C09151=1184.865,-10.764,-44.192,179.961,5.758,149.033
C09152=1184.870,-11.013,-44.179,179.959,5.759,149.034
C09153=1184.875,-11.263,-44.165,179.956,5.758,149.035
C09154=1184.880,-11.512,-44.153,179.953,5.758,149.035
C09155=1184.886,-11.762,-44.139,179.951,5.757,149.036
C09156=1184.891,-12.012,-44.126,179.949,5.756,149.036
C09157=1184.896,-12.261,-44.112,179.946,5.756,149.037
C09158=1184.901,-12.511,-44.099,179.944,5.755,149.038
C09159=1184.907,-12.760,-44.086,179.941,5.755,149.038
C09160=1184.911,-13.010,-44.073,179.938,5.754,149.039
C09161=1184.916,-13.260,-44.061,179.936,5.754,149.040
C09162=1184.922,-13.509,-44.047,179.934,5.754,149.040
C09163=1184.926,-13.759,-44.034,179.932,5.753,149.041
C09164=1184.932,-14.008,-44.021,179.929,5.753,149.041
C09165=1184.937,-14.258,-44.008,179.926,5.752,149.042
C09166=1184.942,-14.508,-43.995,179.924,5.751,149.043
C09167=1184.947,-14.757,-43.981,179.921,5.751,149.043
C09168=1184.952,-15.007,-43.968,179.919,5.751,149.044
C09169=1184.957,-15.256,-43.956,179.916,5.750,149.045
C09170=1184.963,-15.506,-43.942,179.914,5.749,149.045
C09171=1184.967,-15.756,-43.929,179.912,5.750,149.046
C09172=1184.973,-16.005,-43.916,179.909,5.749,149.047
C09173=1184.978,-16.255,-43.903,179.907,5.748,149.047
C09174=1184.983,-16.504,-43.890,179.904,5.748,149.048
C09175=1184.988,-16.754,-43.877,179.902,5.747,149.048
C09176=1184.993,-17.004,-43.864,179.899,5.747,149.049
C09177=1184.998,-17.253,-43.851,179.897,5.746,149.050
C09178=1185.004,-17.503,-43.838,179.894,5.746,149.050
C09179=1185.008,-17.753,-43.825,179.892,5.746,149.051
C09180=1185.014,-18.002,-43.812,179.890,5.745,149.052
C09181=1185.019,-18.251,-43.800,179.887,5.745,149.052
C09182=1185.024,-18.502,-43.786,179.885,5.744,149.053
C09183=1185.029,-18.751,-43.774,179.882,5.744,149.054
C09184=1185.034,-19.000,-43.761,179.880,5.743,149.054
C09185=1185.039,-19.251,-43.747,179.877,5.742,149.055
C09186=1185.045,-19.500,-43.735,179.875,5.742,149.055
C09187=1185.050,-19.749,-43.722,179.872,5.742,149.056
C09188=1185.054,-19.999,-43.709,179.870,5.741,149.057
C09189=1185.060,-20.249,-43.696,179.868,5.741,149.057
C09190=1185.065,-20.498,-43.684,179.865,5.741,149.058
C09191=1185.070,-20.748,-43.671,179.862,5.740,149.059
C09192=1185.075,-20.998,-43.658,179.860,5.739,149.059
C09193=1185.081,-21.247,-43.645,179.857,5.739,149.060
C09194=1185.086,-21.497,-43.632,179.855,5.739,149.060
C09195=1185.090,-21.747,-43.619,179.853,5.739,149.061
C09196=1185.096,-21.996,-43.607,179.851,5.738,149.062
C09197=1185.101,-22.246,-43.593,179.848,5.737,149.062
C09198=1185.106,-22.495,-43.581,179.845,5.737,149.063
C09199=1185.111,-22.745,-43.568,179.843,5.736,149.063
C09200=1185.116,-22.994,-43.555,179.840,5.736,149.064
C09201=1185.122,-23.264,-43.541,179.838,5.735,149.065
C09202=1185.128,-23.534,-43.528,179.835,5.735,149.066
C09203=1185.134,-23.804,-43.514,179.832,5.734,149.066
C09204=1185.139,-24.074,-43.500,179.830,5.734,149.067
C09205=1185.144,-24.323,-43.488,179.828,5.734,149.068
C09206=1185.149,-24.572,-43.475,179.826,5.733,149.068
C09207=1185.154,-24.822,-43.463,179.823,5.733,149.069
C09208=1185.159,-25.072,-43.449,179.820,5.732,149.070
C09209=1185.165,-25.322,-43.437,179.818,5.732,149.070
C09210=1185.170,-25.571,-43.425,179.815,5.731,149.071
C09211=1185.175,-25.820,-43.412,179.813,5.732,149.071
C09212=1185.180,-26.070,-43.399,179.811,5.731,149.072
C09213=1185.184,-26.320,-43.386,179.808,5.731,149.073
C09214=1185.190,-26.569,-43.374,179.806,5.730,149.073
C09215=1185.195,-26.819,-43.362,179.803,5.729,149.074
C09216=1185.201,-27.069,-43.349,179.800,5.729,149.075
C09217=1185.206,-27.318,-43.336,179.799,5.729,149.075
C09218=1185.211,-27.568,-43.323,179.796,5.728,149.076
C09219=1185.216,-27.818,-43.311,179.794,5.728,149.077
C09220=1185.221,-28.067,-43.299,179.791,5.727,149.077
C09221=1185.226,-28.317,-43.286,179.789,5.727,149.078
C09222=1185.231,-28.566,-43.273,179.786,5.726,149.078
C09223=1185.236,-28.817,-43.261,179.784,5.727,149.079
C09224=1185.241,-29.066,-43.249,179.781,5.726,149.080
C09225=1185.246,-29.315,-43.236,179.779,5.725,149.080
C09226=1185.252,-29.565,-43.224,179.776,5.725,149.081
C09227=1185.257,-29.814,-43.212,179.774,5.724,149.082
C09228=1185.262,-30.064,-43.199,179.772,5.725,149.082
C09229=1185.267,-30.314,-43.186,179.770,5.724,149.083
C09230=1185.272,-30.564,-43.174,179.767,5.723,149.084
C09231=1185.277,-30.813,-43.161,179.764,5.723,149.084
C09232=1185.282,-31.062,-43.149,179.762,5.722,149.085
C09233=1185.288,-31.312,-43.137,179.759,5.722,149.085
C09234=1185.293,-31.562,-43.124,179.757,5.722,149.086
C09235=1185.298,-31.812,-43.112,179.755,5.722,149.087
C09236=1185.303,-32.062,-43.100,179.752,5.721,149.087
C09237=1185.308,-32.311,-43.087,179.750,5.720,149.088
C09238=1185.313,-32.561,-43.075,179.747,5.720,149.089
C09239=1185.318,-32.810,-43.062,179.745,5.720,149.089
C09240=1185.324,-33.060,-43.051,179.743,5.719,149.090
C09241=1185.329,-33.309,-43.038,179.740,5.719,149.091
C09242=1185.334,-33.559,-43.025,179.738,5.719,149.091
C09243=1185.340,-33.809,-43.013,179.735,5.718,149.092
C09244=1185.344,-34.059,-43.000,179.733,5.718,149.092
C09245=1185.350,-34.309,-42.989,179.731,5.718,149.093
C09246=1185.355,-34.558,-42.976,179.728,5.717,149.094
C09247=1185.360,-34.808,-42.964,179.726,5.716,149.094
C09248=1185.365,-35.057,-42.952,179.723,5.716,149.095
C09249=1185.371,-35.307,-42.940,179.721,5.716,149.096
C09250=1185.376,-35.556,-42.927,179.718,5.716,149.096
C09251=1185.381,-35.806,-42.915,179.716,5.715,149.097
C09252=1185.386,-36.056,-42.903,179.714,5.715,149.098
C09253=1185.392,-36.306,-42.891,179.712,5.715,149.098
C09254=1185.397,-36.555,-42.878,179.709,5.714,149.099
C09255=1185.402,-36.805,-42.867,179.707,5.714,149.099
C09256=1185.407,-37.054,-42.854,179.704,5.713,149.100
C09257=1185.412,-37.304,-42.842,179.701,5.713,149.101
C09258=1185.417,-37.553,-42.830,179.700,5.713,149.101
C09259=1185.422,-37.804,-42.817,179.697,5.712,149.102
C09260=1185.427,-38.053,-42.805,179.694,5.712,149.103
C09261=1185.433,-38.303,-42.793,179.692,5.711,149.103
C09262=1185.438,-38.552,-42.780,179.690,5.711,149.104
C09263=1185.442,-38.802,-42.769,179.688,5.711,149.105
C09264=1185.448,-39.052,-42.757,179.685,5.710,149.105
C09265=1185.453,-39.301,-42.745,179.683,5.710,149.106
C09266=1185.458,-39.551,-42.733,179.680,5.709,149.106
C09267=1185.464,-39.800,-42.720,179.678,5.710,149.107
C09268=1185.469,-40.050,-42.708,179.675,5.709,149.108
C09269=1185.474,-40.300,-42.697,179.673,5.708,149.108
C09270=1185.479,-40.549,-42.684,179.670,5.708,149.109
C09271=1185.484,-40.799,-42.672,179.668,5.707,149.110
C09272=1185.490,-41.049,-42.661,179.666,5.708,149.110
C09273=1185.495,-41.299,-42.648,179.663,5.707,149.111
C09274=1185.499,-41.548,-42.637,179.661,5.706,149.112
C09275=1185.505,-41.798,-42.625,179.658,5.706,149.112
C09276=1185.510,-42.047,-42.612,179.657,5.706,149.113
C09277=1185.515,-42.297,-42.600,179.654,5.706,149.113
C09278=1185.521,-42.547,-42.588,179.651,5.705,149.114
C09279=1185.525,-42.796,-42.576,179.649,5.705,149.115
C09280=1185.531,-43.046,-42.565,179.647,5.705,149.115
C09281=1185.536,-43.296,-42.553,179.644,5.704,149.116
C09282=1185.541,-43.545,-42.540,179.642,5.704,149.117
C09283=1185.546,-43.795,-42.529,179.639,5.703,149.117
C09284=1185.551,-44.045,-42.517,179.637,5.703,149.118
C09285=1185.557,-44.294,-42.505,179.635,5.703,149.119
C09286=1185.562,-44.543,-42.493,179.632,5.702,149.119
C09287=1185.567,-44.793,-42.481,179.630,5.702,149.120
C09288=1185.573,-45.043,-42.470,179.628,5.702,149.120
C09289=1185.578,-45.293,-42.458,179.625,5.702,149.121
C09290=1185.583,-45.543,-42.446,179.623,5.701,149.122
C09291=1185.588,-45.792,-42.434,179.620,5.700,149.122
C09292=1185.593,-46.042,-42.422,179.618,5.701,149.123
C09293=1185.598,-46.292,-42.411,179.616,5.700,149.124
C09294=1185.603,-46.542,-42.399,179.613,5.699,149.124
C09295=1185.609,-46.791,-42.387,179.611,5.699,149.125
C09296=1185.613,-47.040,-42.375,179.609,5.699,149.126
C09297=1185.619,-47.290,-42.363,179.606,5.699,149.126
C09298=1185.624,-47.540,-42.351,179.604,5.698,149.127
C09299=1185.629,-47.789,-42.340,179.601,5.698,149.127
C09300=1185.635,-48.039,-42.328,179.599,5.698,149.128
C09301=1185.640,-48.289,-42.316,179.597,5.697,149.129
C09302=1185.645,-48.539,-42.305,179.594,5.697,149.129
C09303=1185.650,-48.788,-42.292,179.592,5.696,149.130
C09304=1185.656,-49.038,-42.281,179.589,5.697,149.131
C09305=1185.662,-49.308,-42.269,179.587,5.696,149.131
C09306=1185.667,-49.579,-42.256,179.585,5.695,149.132
C09307=1185.672,-49.849,-42.243,179.582,5.695,149.133
C09308=1185.678,-50.119,-42.230,179.579,5.695,149.133
C09309=1185.683,-50.368,-42.219,179.577,5.694,149.134
C09310=1185.688,-50.618,-42.207,179.575,5.695,149.135
C09311=1185.693,-50.868,-42.196,179.572,5.694,149.135
C09312=1185.699,-51.118,-42.184,179.570,5.693,149.136
C09313=1185.704,-51.368,-42.172,179.568,5.694,149.137
C09314=1185.709,-51.617,-42.161,179.565,5.693,149.137
C09315=1185.715,-51.867,-42.149,179.563,5.692,149.138
C09316=1185.719,-52.116,-42.138,179.560,5.692,149.139
C09317=1185.725,-52.366,-42.126,179.558,5.692,149.139
C09318=1185.729,-52.616,-42.115,179.556,5.692,149.140
C09319=1185.735,-52.866,-42.103,179.553,5.691,149.140
C09320=1185.740,-53.116,-42.091,179.551,5.691,149.141
C09321=1185.746,-53.365,-42.080,179.548,5.691,149.142
C09322=1185.751,-53.615,-42.068,179.546,5.690,149.142
C09323=1185.756,-53.864,-42.057,179.544,5.690,149.143
C09324=1185.761,-54.114,-42.045,179.541,5.690,149.144
C09325=1185.766,-54.364,-42.034,179.539,5.689,149.144
C09326=1185.772,-54.613,-42.022,179.537,5.689,149.145
C09327=1185.777,-54.863,-42.011,179.535,5.689,149.146
C09328=1185.782,-55.112,-41.999,179.532,5.688,149.146
C09329=1185.787,-55.362,-41.988,179.530,5.688,149.147
C09330=1185.792,-55.612,-41.976,179.527,5.688,149.147
C09331=1185.797,-55.862,-41.965,179.525,5.688,149.148
C09332=1185.803,-56.112,-41.954,179.523,5.687,149.149
C09333=1185.808,-56.361,-41.942,179.520,5.687,149.149
C09334=1185.813,-56.611,-41.931,179.518,5.687,149.150
C09335=1185.818,-56.861,-41.919,179.516,5.686,149.151
C09336=1185.823,-57.110,-41.908,179.513,5.686,149.151
C09337=1185.829,-57.360,-41.896,179.511,5.685,149.152
C09338=1185.833,-57.609,-41.885,179.508,5.686,149.153
C09339=1185.839,-57.859,-41.873,179.506,5.685,149.153
C09340=1185.844,-58.109,-41.863,179.504,5.685,149.154
C09341=1185.850,-58.359,-41.851,179.502,5.685,149.155
C09342=1185.855,-58.608,-41.840,179.499,5.684,149.155
C09343=1185.859,-58.858,-41.829,179.497,5.684,149.156
C09344=1185.865,-59.108,-41.817,179.495,5.684,149.156
C09345=1185.870,-59.357,-41.806,179.492,5.683,149.157
C09346=1185.876,-59.607,-41.795,179.490,5.683,149.158
C09347=1185.880,-59.857,-41.783,179.488,5.683,149.158
C09348=1185.886,-60.106,-41.772,179.485,5.683,149.159
C09349=1185.891,-60.356,-41.760,179.483,5.682,149.159
C09350=1185.896,-60.606,-41.750,179.480,5.682,149.160
C09351=1185.902,-60.856,-41.738,179.478,5.682,149.161
C09352=1185.907,-61.105,-41.727,179.476,5.681,149.161
C09353=1185.912,-61.355,-41.716,179.473,5.681,149.162
C09354=1185.917,-61.605,-41.705,179.471,5.681,149.163
C09355=1185.922,-61.855,-41.693,179.469,5.680,149.163
C09356=1185.927,-62.104,-41.682,179.466,5.680,149.164
C09357=1185.933,-62.354,-41.670,179.464,5.680,149.165
C09358=1185.938,-62.604,-41.660,179.462,5.679,149.165
C09359=1185.943,-62.853,-41.649,179.459,5.679,149.166
C09360=1185.948,-63.103,-41.637,179.457,5.679,149.167
C09361=1185.953,-63.353,-41.627,179.455,5.679,149.167
C09362=1185.959,-63.602,-41.616,179.452,5.678,149.168
C09363=1185.964,-63.852,-41.604,179.450,5.678,149.168
C09364=1185.969,-64.101,-41.592,179.448,5.678,149.169
C09365=1185.974,-64.351,-41.582,179.445,5.677,149.170
C09366=1185.980,-64.601,-41.570,179.443,5.678,149.170
C09367=1185.985,-64.851,-41.559,179.441,5.677,149.171
C09368=1185.990,-65.100,-41.549,179.439,5.676,149.172
C09369=1185.996,-65.350,-41.537,179.436,5.677,149.172
C09370=1186.001,-65.600,-41.526,179.434,5.676,149.173
C09371=1186.006,-65.849,-41.515,179.432,5.676,149.173
C09372=1186.011,-66.099,-41.504,179.430,5.676,149.174
C09373=1186.016,-66.349,-41.493,179.427,5.675,149.175
C09374=1186.022,-66.598,-41.482,179.425,5.675,149.175
C09375=1186.027,-66.849,-41.472,179.423,5.675,149.176
C09376=1186.031,-67.098,-41.460,179.420,5.675,149.177
C09377=1186.037,-67.347,-41.449,179.417,5.674,149.177
C09378=1186.042,-67.598,-41.438,179.416,5.674,149.178
C09379=1186.048,-67.847,-41.427,179.413,5.674,149.179
C09380=1186.053,-68.097,-41.417,179.410,5.673,149.179
C09381=1186.058,-68.347,-41.405,179.409,5.673,149.180
C09382=1186.064,-68.596,-41.395,179.406,5.673,149.181
C09383=1186.068,-68.846,-41.383,179.403,5.672,149.181
C09384=1186.074,-69.095,-41.373,179.402,5.672,149.182
C09385=1186.079,-69.345,-41.362,179.399,5.672,149.182
C09386=1186.084,-69.596,-41.351,179.396,5.672,149.183
C09387=1186.090,-69.845,-41.340,179.395,5.672,149.184
C09388=1186.095,-70.095,-41.329,179.392,5.671,149.184
C09389=1186.100,-70.344,-41.318,179.390,5.671,149.185
C09390=1186.105,-70.594,-41.308,179.388,5.671,149.185
C09391=1186.110,-70.844,-41.296,179.385,5.670,149.186
C09392=1186.116,-71.093,-41.285,179.383,5.670,149.187
C09393=1186.121,-71.343,-41.274,179.381,5.670,149.187
C09394=1186.126,-71.593,-41.264,179.378,5.670,149.188
C09395=1186.131,-71.842,-41.253,179.376,5.670,149.189
C09396=1186.137,-72.092,-41.242,179.374,5.669,149.189
C09397=1186.142,-72.342,-41.231,179.371,5.669,149.190
C09398=1186.148,-72.591,-41.220,179.369,5.669,149.191
C09399=1186.152,-72.841,-41.209,179.367,5.668,149.191
C09400=1186.157,-73.091,-41.199,179.364,5.668,149.192
C09401=1186.163,-73.341,-41.188,179.362,5.668,149.193
C09402=1186.168,-73.590,-41.177,179.360,5.667,149.193
C09403=1186.173,-73.840,-41.167,179.357,5.667,149.194
C09404=1186.179,-74.090,-41.155,179.355,5.667,149.194
C09405=1186.184,-74.339,-41.145,179.353,5.667,149.195
C09406=1186.189,-74.590,-41.134,179.351,5.667,149.196
C09407=1186.194,-74.838,-41.123,179.348,5.667,149.196
C09408=1186.199,-75.089,-41.113,179.346,5.666,149.197
C09409=1186.206,-75.359,-41.101,179.344,5.665,149.198
C09410=1186.211,-75.630,-41.090,179.342,5.666,149.198
C09411=1186.216,-75.901,-41.078,179.339,5.665,149.199
C09412=1186.223,-76.172,-41.066,179.336,5.665,149.200
C09413=1186.228,-76.422,-41.056,179.334,5.665,149.200
C09414=1186.233,-76.671,-41.045,179.332,5.664,149.201
C09415=1186.238,-76.922,-41.034,179.329,5.664,149.202
C09416=1186.244,-77.171,-41.024,179.327,5.664,149.202
C09417=1186.249,-77.421,-41.013,179.325,5.664,149.203
C09418=1186.254,-77.670,-41.003,179.322,5.663,149.203
C09419=1186.259,-77.921,-40.992,179.320,5.664,149.204
C09420=1186.264,-78.169,-40.981,179.318,5.663,149.205
C09421=1186.269,-78.420,-40.971,179.316,5.663,149.205
C09422=1186.275,-78.669,-40.960,179.313,5.663,149.206
C09423=1186.280,-78.920,-40.950,179.311,5.662,149.207
C09424=1186.285,-79.168,-40.939,179.309,5.662,149.207
C09425=1186.290,-79.419,-40.928,179.306,5.662,149.208
C09426=1186.296,-79.668,-40.918,179.304,5.661,149.208
C09427=1186.301,-79.918,-40.907,179.302,5.662,149.209
C09428=1186.307,-80.168,-40.897,179.299,5.661,149.210
C09429=1186.312,-80.417,-40.886,179.298,5.661,149.210
C09430=1186.317,-80.667,-40.876,179.295,5.661,149.211
C09431=1186.322,-80.917,-40.866,179.293,5.660,149.212
C09432=1186.327,-81.167,-40.855,179.291,5.660,149.212
C09433=1186.333,-81.417,-40.845,179.288,5.660,149.213
C09434=1186.338,-81.666,-40.833,179.287,5.660,149.213
C09435=1186.343,-81.916,-40.823,179.284,5.660,149.214
C09436=1186.349,-82.165,-40.813,179.281,5.659,149.215
C09437=1186.354,-82.415,-40.803,179.280,5.659,149.215
C09438=1186.359,-82.665,-40.792,179.277,5.659,149.216
C09439=1186.364,-82.915,-40.782,179.275,5.659,149.217
C09440=1186.370,-83.164,-40.771,179.273,5.658,149.217
C09441=1186.374,-83.414,-40.761,179.270,5.658,149.218
C09442=1186.380,-83.664,-40.751,179.268,5.658,149.219
C09443=1186.385,-83.913,-40.740,179.266,5.657,149.219
C09444=1186.390,-84.163,-40.730,179.264,5.658,149.220
C09445=1186.396,-84.413,-40.720,179.262,5.657,149.220
C09446=1186.401,-84.663,-40.709,179.259,5.657,149.221
C09447=1186.406,-84.913,-40.699,179.257,5.657,149.222
C09448=1186.412,-85.162,-40.689,179.255,5.656,149.222
C09449=1186.417,-85.413,-40.678,179.252,5.657,149.223
C09450=1186.422,-85.662,-40.668,179.250,5.656,149.224
C09451=1186.427,-85.911,-40.657,179.248,5.655,149.224
C09452=1186.432,-86.161,-40.647,179.246,5.656,149.225
C09453=1186.438,-86.410,-40.637,179.243,5.655,149.226
C09454=1186.443,-86.661,-40.626,179.241,5.655,149.226
C09455=1186.448,-86.910,-40.616,179.239,5.655,149.227
C09456=1186.454,-87.160,-40.606,179.236,5.654,149.227
C09457=1186.458,-87.410,-40.596,179.234,5.655,149.228
C09458=1186.464,-87.659,-40.586,179.232,5.654,149.229
C09459=1186.469,-87.909,-40.575,179.230,5.654,149.229
C09460=1186.474,-88.159,-40.565,179.227,5.654,149.230
C09461=1186.480,-88.409,-40.555,179.225,5.653,149.231
C09462=1186.486,-88.658,-40.544,179.223,5.653,149.231
C09463=1186.490,-88.908,-40.534,179.220,5.653,149.232
C09464=1186.495,-89.158,-40.524,179.219,5.653,149.232
C09465=1186.501,-89.407,-40.514,179.216,5.653,149.233
C09466=1186.506,-89.657,-40.503,179.214,5.653,149.234
C09467=1186.512,-89.907,-40.493,179.212,5.652,149.234
C09468=1186.517,-90.156,-40.484,179.209,5.652,149.235
C09469=1186.522,-90.407,-40.474,179.207,5.652,149.236
C09470=1186.527,-90.657,-40.463,179.205,5.651,149.236
C09471=1186.533,-90.906,-40.453,179.203,5.652,149.237
C09472=1186.537,-91.156,-40.443,179.201,5.651,149.237
C09473=1186.543,-91.406,-40.433,179.198,5.651,149.238
C09474=1186.548,-91.655,-40.423,179.196,5.651,149.239
C09475=1186.553,-91.905,-40.412,179.194,5.650,149.239
C09476=1186.558,-92.155,-40.403,179.192,5.651,149.240
C09477=1186.564,-92.404,-40.392,179.189,5.650,149.241
C09478=1186.570,-92.654,-40.382,179.187,5.650,149.241
C09479=1186.575,-92.905,-40.372,179.185,5.650,149.242
C09480=1186.580,-93.154,-40.363,179.183,5.649,149.242
C09481=1186.585,-93.403,-40.353,179.180,5.649,149.243
C09482=1186.590,-93.654,-40.342,179.178,5.649,149.244
C09483=1186.596,-93.903,-40.332,179.176,5.649,149.244
C09484=1186.601,-94.152,-40.322,179.173,5.649,149.245
C09485=1186.607,-94.403,-40.313,179.172,5.649,149.245
C09486=1186.612,-94.653,-40.302,179.169,5.648,149.246
C09487=1186.617,-94.902,-40.293,179.167,5.649,149.247
C09488=1186.622,-95.152,-40.282,179.165,5.648,149.247
C09489=1186.628,-95.401,-40.272,179.162,5.647,149.248
C09490=1186.632,-95.652,-40.263,179.161,5.647,149.248
C09491=1186.638,-95.901,-40.253,179.158,5.647,149.249
C09492=1186.643,-96.151,-40.242,179.156,5.647,149.250
C09493=1186.648,-96.400,-40.233,179.154,5.647,149.250
C09494=1186.653,-96.650,-40.222,179.152,5.647,149.251
C09495=1186.659,-96.900,-40.213,179.149,5.646,149.252
C09496=1186.664,-97.150,-40.203,179.147,5.646,149.252
C09497=1186.670,-97.399,-40.193,179.145,5.646,149.253
C09498=1186.675,-97.649,-40.183,179.143,5.645,149.253
C09499=1186.680,-97.899,-40.173,179.140,5.646,149.254
C09500=1186.685,-98.149,-40.163,179.138,5.645,149.255
C09501=1186.691,-98.398,-40.153,179.136,5.645,149.255
C09502=1186.696,-98.648,-40.144,179.133,5.645,149.256
C09503=1186.702,-98.898,-40.134,179.132,5.645,149.257
C09504=1186.707,-99.148,-40.123,179.129,5.645,149.257
C09505=1186.712,-99.397,-40.114,179.127,5.644,149.258
C09506=1186.718,-99.647,-40.104,179.125,5.644,149.258
C09507=1186.722,-99.897,-40.095,179.122,5.644,149.259
C09508=1186.728,-100.146,-40.084,179.121,5.644,149.260
C09509=1186.733,-100.397,-40.075,179.118,5.643,149.260
C09510=1186.738,-100.646,-40.065,179.116,5.643,149.261
C09511=1186.744,-100.896,-40.055,179.114,5.643,149.262
C09512=1186.749,-101.146,-40.046,179.112,5.643,149.262
C09513=1186.755,-101.417,-40.034,179.109,5.643,149.263
C09514=1186.760,-101.689,-40.024,179.107,5.642,149.264
C09515=1186.766,-101.960,-40.014,179.105,5.643,149.264
C09516=1186.772,-102.232,-40.003,179.102,5.642,149.265
C09517=1186.778,-102.482,-39.994,179.100,5.641,149.265
C09518=1186.782,-102.732,-39.984,179.098,5.642,149.266
C09519=1186.787,-102.981,-39.974,179.096,5.641,149.267
C09520=1186.793,-103.232,-39.964,179.093,5.642,149.267
C09521=1186.798,-103.481,-39.954,179.091,5.641,149.268
C09522=1186.804,-103.731,-39.945,179.089,5.641,149.269
C09523=1186.809,-103.980,-39.935,179.086,5.641,149.269
C09524=1186.815,-104.230,-39.926,179.085,5.641,149.270
C09525=1186.819,-104.480,-39.916,179.082,5.640,149.270
C09526=1186.825,-104.730,-39.906,179.081,5.640,149.271
C09527=1186.830,-104.980,-39.897,179.078,5.640,149.272
C09528=1186.835,-105.229,-39.887,179.076,5.640,149.272
C09529=1186.841,-105.479,-39.878,179.074,5.640,149.273
C09530=1186.846,-105.729,-39.867,179.071,5.639,149.274
C09531=1186.851,-105.978,-39.859,179.069,5.639,149.274
C09532=1186.857,-106.228,-39.848,179.067,5.639,149.275
C09533=1186.862,-106.478,-39.839,179.065,5.639,149.275
C09534=1186.866,-106.728,-39.830,179.062,5.638,149.276
C09535=1186.872,-106.978,-39.820,179.060,5.639,149.277
C09536=1186.877,-107.227,-39.810,179.058,5.638,149.277
C09537=1186.883,-107.477,-39.801,179.056,5.638,149.278
C09538=1186.888,-107.727,-39.791,179.054,5.638,149.278
C09539=1186.894,-107.977,-39.782,179.052,5.638,149.279
C09540=1186.899,-108.226,-39.772,179.050,5.637,149.280
C09541=1186.905,-108.476,-39.763,179.048,5.638,149.280
C09542=1186.910,-108.726,-39.754,179.045,5.637,149.281
C09543=1186.915,-108.975,-39.744,179.043,5.637,149.281
C09544=1186.921,-109.225,-39.735,179.041,5.637,149.282
C09545=1186.925,-109.475,-39.725,179.039,5.637,149.283
C09546=1186.931,-109.725,-39.715,179.036,5.637,149.283
C09547=1186.936,-109.975,-39.706,179.035,5.637,149.284
C09548=1186.941,-110.225,-39.697,179.032,5.636,149.285
C09549=1186.947,-110.475,-39.687,179.030,5.636,149.285
C09550=1186.952,-110.724,-39.678,179.028,5.636,149.286
C09551=1186.957,-110.974,-39.668,179.026,5.635,149.286
C09552=1186.962,-111.223,-39.658,179.023,5.635,149.287
C09553=1186.967,-111.473,-39.650,179.021,5.635,149.287
C09554=1186.973,-111.723,-39.640,179.019,5.635,149.288
C09555=1186.978,-111.973,-39.630,179.017,5.634,149.289
C09556=1186.984,-112.223,-39.621,179.015,5.635,149.289
C09557=1186.989,-112.473,-39.612,179.012,5.634,149.290
C09558=1186.994,-112.722,-39.602,179.011,5.634,149.291
C09559=1187.000,-112.972,-39.593,179.008,5.634,149.291
C09560=1187.005,-113.222,-39.584,179.006,5.634,149.292
C09561=1187.010,-113.471,-39.574,179.004,5.634,149.292
C09562=1187.016,-113.721,-39.565,179.002,5.634,149.293
C09563=1187.021,-113.971,-39.556,178.999,5.633,149.294
C09564=1187.026,-114.220,-39.546,178.998,5.633,149.294
C09565=1187.032,-114.470,-39.537,178.995,5.633,149.295
C09566=1187.037,-114.720,-39.528,178.994,5.633,149.295
C09567=1187.042,-114.970,-39.519,178.991,5.632,149.296
C09568=1187.048,-115.220,-39.509,178.989,5.632,149.297
C09569=1187.053,-115.470,-39.500,178.987,5.632,149.297
C09570=1187.058,-115.719,-39.491,178.985,5.632,149.298
C09571=1187.063,-115.969,-39.482,178.982,5.632,149.298
C09572=1187.069,-116.219,-39.472,178.981,5.632,149.299
C09573=1187.074,-116.469,-39.463,178.978,5.631,149.300
C09574=1187.079,-116.719,-39.454,178.976,5.632,149.300
C09575=1187.085,-116.969,-39.445,178.974,5.631,149.301
C09576=1187.090,-117.218,-39.435,178.972,5.631,149.302
C09577=1187.095,-117.468,-39.426,178.969,5.631,149.302
C09578=1187.100,-117.718,-39.417,178.967,5.631,149.303
C09579=1187.106,-117.968,-39.408,178.965,5.630,149.303
C09580=1187.111,-118.218,-39.399,178.963,5.631,149.304
C09581=1187.116,-118.467,-39.389,178.961,5.630,149.304
C09582=1187.121,-118.717,-39.380,178.959,5.630,149.305
C09583=1187.127,-118.967,-39.371,178.957,5.629,149.306
C09584=1187.133,-119.216,-39.362,178.955,5.630,149.306
C09585=1187.138,-119.466,-39.354,178.952,5.629,149.307
C09586=1187.143,-119.716,-39.345,178.950,5.629,149.308
C09587=1187.148,-119.965,-39.335,178.948,5.629,149.308
C09588=1187.154,-120.215,-39.326,178.946,5.629,149.309
C09589=1187.159,-120.465,-39.317,178.944,5.628,149.309
C09590=1187.165,-120.715,-39.308,178.942,5.629,149.310
C09591=1187.170,-120.965,-39.299,178.940,5.628,149.311
C09592=1187.175,-121.215,-39.290,178.937,5.628,149.311
C09593=1187.181,-121.465,-39.280,178.936,5.628,149.312
C09594=1187.186,-121.715,-39.272,178.933,5.628,149.312
C09595=1187.191,-121.964,-39.262,178.932,5.628,149.313
C09596=1187.196,-122.214,-39.253,178.929,5.628,149.314
C09597=1187.202,-122.463,-39.245,178.927,5.628,149.314
C09598=1187.207,-122.713,-39.236,178.925,5.627,149.315
C09599=1187.213,-122.963,-39.226,178.923,5.627,149.315
C09600=1187.218,-123.213,-39.217,178.920,5.627,149.316
C09601=1187.223,-123.462,-39.208,178.919,5.627,149.317
C09602=1187.228,-123.712,-39.199,178.916,5.627,149.317
C09603=1187.234,-123.962,-39.191,178.914,5.627,149.318
C09604=1187.239,-124.212,-39.182,178.912,5.626,149.318
C09605=1187.245,-124.462,-39.172,178.910,5.626,149.319
C09606=1187.250,-124.711,-39.164,178.908,5.625,149.319
C09607=1187.256,-124.961,-39.155,178.906,5.626,149.320
C09608=1187.261,-125.211,-39.146,178.904,5.625,149.321
C09609=1187.266,-125.461,-39.137,178.902,5.625,149.321
C09610=1187.271,-125.711,-39.128,178.899,5.625,149.322
C09611=1187.276,-125.961,-39.119,178.897,5.625,149.323
C09612=1187.281,-126.210,-39.110,178.895,5.624,149.323
C09613=1187.287,-126.460,-39.102,178.893,5.625,149.324
C09614=1187.293,-126.710,-39.092,178.891,5.624,149.324
C09615=1187.298,-126.960,-39.083,178.889,5.624,149.325
C09616=1187.303,-127.209,-39.074,178.887,5.624,149.325
C09617=1186.881,-127.220,-39.114,178.883,5.628,149.327
C09618=1186.876,-126.970,-39.123,178.885,5.628,149.327
C09619=1186.871,-126.720,-39.132,178.888,5.628,149.326
C09620=1186.866,-126.471,-39.140,178.889,5.628,149.326
C09621=1186.861,-126.221,-39.149,178.892,5.628,149.325
C09622=1186.855,-125.971,-39.158,178.893,5.628,149.324
C09623=1186.850,-125.722,-39.167,178.895,5.628,149.324
C09624=1186.845,-125.472,-39.176,178.898,5.629,149.323
C09625=1186.839,-125.222,-39.185,178.899,5.629,149.323
C09626=1186.833,-124.972,-39.194,178.902,5.629,149.322
C09627=1186.828,-124.722,-39.203,178.904,5.629,149.321
C09628=1186.823,-124.472,-39.212,178.906,5.629,149.321
C09629=1186.818,-124.222,-39.221,178.908,5.629,149.320
C09630=1186.812,-123.973,-39.229,178.911,5.630,149.320
C09631=1186.807,-123.723,-39.238,178.912,5.630,149.319
C09632=1186.802,-123.473,-39.247,178.915,5.630,149.318
C09633=1186.796,-123.223,-39.257,178.916,5.630,149.318
C09634=1186.791,-122.974,-39.266,178.919,5.631,149.317
C09635=1186.786,-122.724,-39.275,178.921,5.631,149.317
C09636=1186.781,-122.474,-39.284,178.923,5.631,149.316
C09637=1186.776,-122.225,-39.293,178.925,5.631,149.315
C09638=1186.770,-121.975,-39.302,178.928,5.631,149.315
C09639=1186.765,-121.724,-39.311,178.929,5.631,149.314
C09640=1186.759,-121.475,-39.320,178.932,5.632,149.314
C09641=1186.754,-121.225,-39.329,178.934,5.632,149.313
C09642=1186.748,-120.976,-39.338,178.936,5.632,149.312
C09643=1186.743,-120.726,-39.346,178.938,5.632,149.312
C09644=1186.737,-120.476,-39.356,178.940,5.632,149.311
C09645=1186.733,-120.226,-39.366,178.942,5.632,149.311
C09646=1186.727,-119.977,-39.374,178.945,5.633,149.310
C09647=1186.722,-119.727,-39.383,178.946,5.633,149.309
C09648=1186.717,-119.477,-39.392,178.949,5.633,149.309
C09649=1186.711,-119.227,-39.402,178.951,5.633,149.308
C09650=1186.706,-118.977,-39.411,178.953,5.633,149.308
C09651=1186.701,-118.728,-39.420,178.955,5.633,149.307
C09652=1186.696,-118.478,-39.429,178.958,5.634,149.306
C09653=1186.691,-118.228,-39.438,178.959,5.634,149.306
C09654=1186.684,-117.978,-39.447,178.962,5.634,149.305
C09655=1186.679,-117.729,-39.456,178.963,5.634,149.305
C09656=1186.674,-117.479,-39.466,178.966,5.635,149.304
C09657=1186.669,-117.230,-39.475,178.968,5.635,149.303
C09658=1186.663,-116.979,-39.484,178.970,5.635,149.303
C09659=1186.658,-116.729,-39.493,178.972,5.635,149.302
C09660=1186.653,-116.480,-39.502,178.975,5.635,149.302
C09661=1186.647,-116.230,-39.512,178.976,5.635,149.301
C09662=1186.642,-115.980,-39.521,178.979,5.636,149.300
C09663=1186.637,-115.730,-39.530,178.981,5.636,149.300
C09664=1186.632,-115.481,-39.539,178.983,5.636,149.299
C09665=1186.626,-115.231,-39.549,178.985,5.636,149.299
C09666=1186.621,-114.981,-39.558,178.988,5.636,149.298
C09667=1186.616,-114.731,-39.567,178.989,5.636,149.297
C09668=1186.610,-114.481,-39.576,178.992,5.637,149.297
C09669=1186.605,-114.232,-39.586,178.993,5.637,149.296
C09670=1186.600,-113.982,-39.595,178.996,5.637,149.296
C09671=1186.594,-113.732,-39.604,178.998,5.637,149.295
C09672=1186.589,-113.483,-39.614,179.000,5.638,149.294
C09673=1186.584,-113.233,-39.623,179.002,5.637,149.294
C09674=1186.578,-112.983,-39.632,179.005,5.638,149.293
C09675=1186.573,-112.733,-39.642,179.007,5.637,149.292
C09676=1186.568,-112.484,-39.651,179.009,5.638,149.292
C09677=1186.562,-112.233,-39.660,179.011,5.638,149.291
C09678=1186.557,-111.984,-39.670,179.013,5.639,149.291
C09679=1186.552,-111.734,-39.679,179.015,5.638,149.290
C09680=1186.546,-111.484,-39.688,179.017,5.639,149.290
C09681=1186.541,-111.235,-39.698,179.020,5.639,149.289
C09682=1186.535,-110.985,-39.707,179.022,5.639,149.288
C09683=1186.530,-110.735,-39.716,179.024,5.639,149.288
C09684=1186.525,-110.486,-39.726,179.026,5.640,149.287
C09685=1186.519,-110.236,-39.735,179.028,5.639,149.286
C09686=1186.515,-109.986,-39.745,179.030,5.640,149.286
C09687=1186.509,-109.735,-39.755,179.032,5.640,149.285
C09688=1186.504,-109.486,-39.764,179.035,5.640,149.285
C09689=1186.499,-109.236,-39.773,179.037,5.640,149.284
C09690=1186.493,-108.986,-39.783,179.039,5.640,149.283
C09691=1186.489,-108.737,-39.793,179.041,5.640,149.283
C09692=1186.483,-108.487,-39.802,179.044,5.641,149.282
C09693=1186.478,-108.238,-39.812,179.045,5.641,149.282
C09694=1186.472,-107.987,-39.821,179.048,5.641,149.281
C09695=1186.467,-107.738,-39.830,179.049,5.641,149.280
C09696=1186.462,-107.488,-39.840,179.052,5.642,149.280
C09697=1186.456,-107.238,-39.849,179.054,5.642,149.279
C09698=1186.451,-106.989,-39.859,179.056,5.642,149.279
C09699=1186.445,-106.739,-39.868,179.059,5.642,149.278
C09700=1186.441,-106.489,-39.878,179.061,5.642,149.277
C09701=1186.435,-106.239,-39.888,179.063,5.643,149.277
C09702=1186.430,-105.989,-39.897,179.065,5.643,149.276
C09703=1186.424,-105.739,-39.907,179.068,5.643,149.275
C09704=1186.419,-105.490,-39.916,179.069,5.643,149.275
C09705=1186.413,-105.240,-39.926,179.072,5.644,149.274
C09706=1186.409,-104.991,-39.936,179.074,5.643,149.273
C09707=1186.403,-104.740,-39.945,179.076,5.644,149.273
C09708=1186.398,-104.491,-39.955,179.078,5.644,149.272
C09709=1186.393,-104.241,-39.965,179.080,5.644,149.272
C09710=1186.388,-103.991,-39.974,179.083,5.644,149.271
C09711=1186.382,-103.742,-39.984,179.085,5.645,149.271
C09712=1186.377,-103.492,-39.993,179.087,5.644,149.270
C09713=1186.371,-103.242,-40.003,179.089,5.645,149.269
C09714=1186.366,-102.992,-40.012,179.092,5.645,149.269
C09715=1186.361,-102.743,-40.023,179.094,5.645,149.268
C09716=1186.356,-102.493,-40.033,179.096,5.646,149.267
C09717=1186.350,-102.243,-40.042,179.098,5.645,149.267
C09718=1186.345,-101.971,-40.053,179.101,5.646,149.266
C09719=1186.339,-101.700,-40.063,179.103,5.647,149.266
C09720=1186.333,-101.428,-40.074,179.105,5.646,149.265
C09721=1186.328,-101.157,-40.085,179.108,5.647,149.264
C09722=1186.323,-100.907,-40.093,179.110,5.646,149.263
C09723=1186.317,-100.657,-40.104,179.112,5.647,149.263
C09724=1186.311,-100.408,-40.114,179.115,5.647,149.262
C09725=1186.307,-100.157,-40.123,179.116,5.647,149.262
C09726=1186.301,-99.908,-40.133,179.119,5.648,149.261
C09727=1186.296,-99.658,-40.143,179.121,5.648,149.261
C09728=1186.290,-99.408,-40.152,179.123,5.648,149.260
C09729=1186.285,-99.159,-40.163,179.125,5.648,149.259
C09730=1186.281,-98.909,-40.173,179.127,5.649,149.259
C09731=1186.275,-98.659,-40.182,179.130,5.648,149.258
C09732=1186.270,-98.409,-40.192,179.132,5.649,149.257
C09733=1186.264,-98.160,-40.202,179.134,5.649,149.257
C09734=1186.259,-97.910,-40.212,179.137,5.649,149.256
C09735=1186.254,-97.660,-40.221,179.139,5.650,149.256
C09736=1186.248,-97.410,-40.232,179.141,5.649,149.255
C09737=1186.243,-97.161,-40.242,179.143,5.650,149.254
C09738=1186.238,-96.911,-40.251,179.145,5.650,149.254
C09739=1186.232,-96.661,-40.261,179.148,5.650,149.253
C09740=1186.227,-96.411,-40.272,179.149,5.650,149.252
C09741=1186.222,-96.162,-40.281,179.152,5.651,149.252
C09742=1186.217,-95.912,-40.291,179.154,5.651,149.251
C09743=1186.211,-95.662,-40.301,179.156,5.651,149.251
C09744=1186.206,-95.412,-40.311,179.159,5.651,149.250
C09745=1186.201,-95.163,-40.321,179.161,5.651,149.249
C09746=1186.195,-94.913,-40.331,179.163,5.652,149.249
C09747=1186.190,-94.663,-40.340,179.165,5.652,149.248
C09748=1186.185,-94.413,-40.351,179.167,5.652,149.247
C09749=1186.179,-94.163,-40.361,179.170,5.652,149.247
C09750=1186.175,-93.914,-40.371,179.172,5.653,149.246
C09751=1186.169,-93.665,-40.381,179.174,5.653,149.246
C09752=1186.164,-93.414,-40.391,179.176,5.653,149.245
C09753=1186.158,-93.164,-40.401,179.179,5.653,149.244
C09754=1186.153,-92.915,-40.410,179.181,5.653,149.244
C09755=1186.148,-92.665,-40.421,179.183,5.654,149.243
C09756=1186.143,-92.415,-40.431,179.185,5.653,149.242
C09757=1186.137,-92.166,-40.441,179.187,5.654,149.242
C09758=1186.132,-91.916,-40.451,179.190,5.655,149.241
C09759=1186.127,-91.666,-40.462,179.192,5.654,149.241
C09760=1186.122,-91.417,-40.472,179.194,5.655,149.240
C09761=1186.116,-91.166,-40.481,179.196,5.655,149.239
C09762=1186.111,-90.917,-40.491,179.198,5.655,149.239
C09763=1186.106,-90.667,-40.502,179.201,5.655,149.238
C09764=1186.100,-90.417,-40.512,179.203,5.655,149.237
C09765=1186.095,-90.168,-40.522,179.205,5.656,149.237
C09766=1186.090,-89.918,-40.532,179.207,5.656,149.236
C09767=1186.085,-89.668,-40.542,179.210,5.656,149.236
C09768=1186.079,-89.419,-40.552,179.212,5.656,149.235
C09769=1186.074,-89.169,-40.563,179.214,5.657,149.234
C09770=1186.069,-88.919,-40.573,179.217,5.657,149.234
C09771=1186.064,-88.670,-40.583,179.219,5.657,149.233
C09772=1186.059,-88.420,-40.593,179.221,5.657,149.232
C09773=1186.053,-88.170,-40.604,179.223,5.657,149.232
C09774=1186.048,-87.921,-40.614,179.226,5.658,149.231
C09775=1186.043,-87.670,-40.624,179.228,5.657,149.231
C09776=1186.037,-87.421,-40.635,179.230,5.658,149.230
C09777=1186.032,-87.172,-40.644,179.233,5.659,149.229
C09778=1186.027,-86.921,-40.655,179.234,5.659,149.229
C09779=1186.021,-86.672,-40.665,179.237,5.659,149.228
C09780=1186.016,-86.421,-40.675,179.239,5.659,149.227
C09781=1186.011,-86.172,-40.686,179.241,5.659,149.227
C09782=1186.005,-85.922,-40.696,179.244,5.660,149.226
C09783=1186.001,-85.672,-40.706,179.246,5.659,149.226
C09784=1185.995,-85.423,-40.716,179.248,5.660,149.225
C09785=1185.990,-85.173,-40.726,179.250,5.660,149.224
C09786=1185.985,-84.923,-40.737,179.252,5.661,149.224
C09787=1185.979,-84.674,-40.747,179.255,5.661,149.223
C09788=1185.974,-84.423,-40.758,179.257,5.661,149.222
C09789=1185.969,-84.174,-40.769,179.259,5.661,149.222
C09790=1185.963,-83.925,-40.779,179.261,5.661,149.221
C09791=1185.958,-83.675,-40.789,179.264,5.661,149.221
C09792=1185.953,-83.425,-40.799,179.266,5.662,149.220
C09793=1185.948,-83.175,-40.810,179.268,5.662,149.219
C09794=1185.943,-82.926,-40.820,179.271,5.662,149.219
C09795=1185.937,-82.676,-40.830,179.273,5.662,149.218
C09796=1185.932,-82.426,-40.841,179.275,5.663,149.217
C09797=1185.927,-82.177,-40.851,179.277,5.663,149.217
C09798=1185.922,-81.927,-40.862,179.280,5.663,149.216
C09799=1185.916,-81.677,-40.872,179.282,5.663,149.216
C09800=1185.911,-81.427,-40.883,179.284,5.663,149.215
C09801=1185.906,-81.177,-40.893,179.286,5.664,149.214
C09802=1185.900,-80.928,-40.903,179.289,5.664,149.214
C09803=1185.896,-80.678,-40.915,179.291,5.664,149.213
C09804=1185.890,-80.429,-40.925,179.293,5.665,149.212
C09805=1185.885,-80.178,-40.935,179.296,5.665,149.212
C09806=1185.879,-79.929,-40.946,179.298,5.665,149.211
C09807=1185.874,-79.679,-40.956,179.300,5.666,149.211
C09808=1185.869,-79.430,-40.967,179.302,5.665,149.210
C09809=1185.864,-79.179,-40.978,179.305,5.666,149.209
C09810=1185.858,-78.930,-40.988,179.307,5.666,149.209
C09811=1185.853,-78.680,-40.998,179.309,5.666,149.208
C09812=1185.848,-78.431,-41.009,179.312,5.667,149.207
C09813=1185.843,-78.181,-41.020,179.314,5.666,149.207
C09814=1185.838,-77.931,-41.030,179.316,5.667,149.206
C09815=1185.832,-77.681,-41.040,179.319,5.668,149.206
C09816=1185.827,-77.432,-41.052,179.321,5.667,149.205
C09817=1185.822,-77.182,-41.062,179.323,5.668,149.204
C09818=1185.817,-76.932,-41.072,179.325,5.668,149.204
C09819=1185.811,-76.683,-41.083,179.328,5.668,149.203
C09820=1185.806,-76.433,-41.094,179.330,5.669,149.202
C09821=1185.801,-76.183,-41.104,179.332,5.668,149.202
C09822=1185.795,-75.912,-41.116,179.334,5.669,149.201
C09823=1185.790,-75.641,-41.127,179.337,5.669,149.200
C09824=1185.784,-75.371,-41.139,179.340,5.670,149.200
C09825=1185.778,-75.099,-41.151,179.342,5.670,149.199
C09826=1185.773,-74.850,-41.162,179.344,5.670,149.198
C09827=1185.768,-74.600,-41.172,179.347,5.671,149.198
C09828=1185.762,-74.350,-41.182,179.349,5.670,149.197
C09829=1185.757,-74.101,-41.194,179.351,5.671,149.197
C09830=1185.752,-73.850,-41.204,179.354,5.671,149.196
C09831=1185.747,-73.602,-41.215,179.356,5.671,149.195
C09832=1185.741,-73.351,-41.226,179.358,5.672,149.195
C09833=1185.736,-73.101,-41.237,179.361,5.672,149.194
C09834=1185.731,-72.852,-41.248,179.363,5.672,149.193
C09835=1185.725,-72.602,-41.258,179.365,5.673,149.193
C09836=1185.721,-72.353,-41.269,179.368,5.673,149.192
C09837=1185.715,-72.103,-41.280,179.370,5.673,149.191
C09838=1185.710,-71.853,-41.290,179.372,5.673,149.191
C09839=1185.704,-71.604,-41.302,179.375,5.674,149.190
C09840=1185.699,-71.353,-41.312,179.377,5.673,149.189
C09841=1185.694,-71.104,-41.324,179.379,5.674,149.189
C09842=1185.689,-70.854,-41.334,179.381,5.674,149.188
C09843=1185.684,-70.605,-41.345,179.384,5.674,149.188
C09844=1185.678,-70.355,-41.355,179.386,5.675,149.187
C09845=1185.673,-70.105,-41.367,179.388,5.675,149.186
C09846=1185.667,-69.856,-41.377,179.390,5.675,149.186
C09847=1185.663,-69.606,-41.389,179.393,5.676,149.185
C09848=1185.658,-69.356,-41.399,179.395,5.676,149.184
C09849=1185.652,-69.107,-41.410,179.397,5.676,149.184
C09850=1185.647,-68.856,-41.421,179.400,5.677,149.183
C09851=1185.641,-68.607,-41.432,179.402,5.676,149.183
C09852=1185.636,-68.357,-41.443,179.404,5.677,149.182
C09853=1185.632,-68.107,-41.454,179.407,5.678,149.181
C09854=1185.626,-67.858,-41.464,179.409,5.677,149.181
C09855=1185.621,-67.608,-41.476,179.411,5.678,149.180
C09856=1185.615,-67.359,-41.487,179.413,5.679,149.180
C09857=1185.610,-67.109,-41.498,179.416,5.678,149.179
C09858=1185.606,-66.859,-41.509,179.418,5.679,149.178
C09859=1185.599,-66.609,-41.520,179.420,5.679,149.178
C09860=1185.595,-66.360,-41.531,179.422,5.679,149.177
C09861=1185.590,-66.109,-41.542,179.425,5.679,149.176
C09862=1185.584,-65.861,-41.553,179.428,5.680,149.175
C09863=1185.579,-65.611,-41.564,179.429,5.680,149.175
C09864=1185.574,-65.360,-41.575,179.432,5.680,149.174
C09865=1185.569,-65.111,-41.586,179.435,5.681,149.174
C09866=1185.563,-64.861,-41.598,179.436,5.681,149.173
C09867=1185.558,-64.611,-41.608,179.439,5.681,149.172
C09868=1185.553,-64.362,-41.619,179.442,5.682,149.172
C09869=1185.548,-64.112,-41.631,179.443,5.682,149.171
C09870=1185.543,-63.862,-41.642,179.446,5.682,149.171
C09871=1185.537,-63.613,-41.653,179.449,5.682,149.170
C09872=1185.533,-63.364,-41.664,179.450,5.682,149.169
C09873=1185.527,-63.113,-41.675,179.453,5.683,149.169
C09874=1185.522,-62.864,-41.686,179.456,5.683,149.168
C09875=1185.517,-62.614,-41.697,179.457,5.683,149.167
C09876=1185.511,-62.364,-41.709,179.460,5.684,149.167
C09877=1185.506,-62.115,-41.719,179.462,5.684,149.166
C09878=1185.501,-61.865,-41.731,179.465,5.684,149.165
C09879=1185.496,-61.615,-41.743,179.467,5.685,149.165
C09880=1185.490,-61.366,-41.753,179.469,5.685,149.164
C09881=1185.485,-61.116,-41.765,179.471,5.685,149.163
C09882=1185.480,-60.866,-41.776,179.474,5.685,149.163
C09883=1185.475,-60.617,-41.787,179.476,5.686,149.162
C09884=1185.469,-60.367,-41.798,179.479,5.686,149.162
C09885=1185.464,-60.117,-41.809,179.481,5.686,149.161
C09886=1185.460,-59.868,-41.821,179.483,5.687,149.160
C09887=1185.454,-59.618,-41.833,179.486,5.687,149.160
C09888=1185.449,-59.368,-41.843,179.488,5.687,149.159
C09889=1185.443,-59.118,-41.855,179.490,5.688,149.159
C09890=1185.438,-58.869,-41.866,179.493,5.688,149.158
C09891=1185.433,-58.620,-41.877,179.495,5.688,149.157
C09892=1185.428,-58.370,-41.889,179.497,5.688,149.157
C09893=1185.423,-58.120,-41.900,179.500,5.689,149.156
C09894=1185.417,-57.869,-41.911,179.502,5.688,149.155
C09895=1185.413,-57.620,-41.923,179.504,5.689,149.155
C09896=1185.407,-57.371,-41.934,179.507,5.690,149.154
C09897=1185.402,-57.121,-41.945,179.509,5.690,149.153
C09898=1185.397,-56.871,-41.957,179.511,5.690,149.153
C09899=1185.392,-56.621,-41.969,179.514,5.691,149.152
C09900=1185.386,-56.373,-41.979,179.516,5.691,149.151
C09901=1185.381,-56.122,-41.991,179.518,5.691,149.151
C09902=1185.376,-55.872,-42.002,179.521,5.691,149.150
C09903=1185.371,-55.622,-42.014,179.523,5.692,149.150
C09904=1185.366,-55.373,-42.025,179.526,5.692,149.149
C09905=1185.360,-55.124,-42.037,179.527,5.692,149.148
C09906=1185.355,-54.874,-42.048,179.530,5.693,149.148
C09907=1185.350,-54.624,-42.060,179.533,5.693,149.147
C09908=1185.345,-54.374,-42.071,179.534,5.693,149.146
C09909=1185.340,-54.124,-42.083,179.537,5.694,149.146
C09910=1185.334,-53.876,-42.094,179.540,5.694,149.145
C09911=1185.329,-53.626,-42.106,179.542,5.694,149.144
C09912=1185.324,-53.376,-42.117,179.544,5.695,149.144
C09913=1185.319,-53.126,-42.129,179.547,5.695,149.143
C09914=1185.314,-52.876,-42.140,179.549,5.695,149.142
C09915=1185.309,-52.626,-42.152,179.551,5.695,149.142
C09916=1185.303,-52.378,-42.163,179.554,5.696,149.141
C09917=1185.298,-52.128,-42.175,179.556,5.696,149.141
C09918=1185.292,-51.878,-42.187,179.559,5.697,149.140
C09919=1185.288,-51.628,-42.198,179.561,5.697,149.139
C09920=1185.282,-51.378,-42.210,179.563,5.697,149.139
C09921=1185.278,-51.128,-42.221,179.566,5.698,149.138
C09922=1185.272,-50.879,-42.233,179.567,5.698,149.138
C09923=1185.267,-50.630,-42.244,179.570,5.698,149.137
C09924=1185.262,-50.380,-42.256,179.573,5.698,149.136
C09925=1185.256,-50.130,-42.268,179.575,5.699,149.136
C09926=1185.251,-49.859,-42.281,179.578,5.700,149.135
C09927=1185.245,-49.590,-42.293,179.580,5.699,149.134
C09928=1185.239,-49.319,-42.306,179.582,5.700,149.134
C09929=1185.234,-49.048,-42.319,179.585,5.700,149.133
C09930=1185.229,-48.799,-42.330,179.588,5.701,149.132
C09931=1185.223,-48.550,-42.341,179.590,5.701,149.131
C09932=1185.218,-48.300,-42.353,179.592,5.701,149.131
C09933=1185.213,-48.050,-42.365,179.595,5.702,149.130
C09934=1185.208,-47.801,-42.377,179.597,5.702,149.130
C09935=1185.203,-47.551,-42.388,179.600,5.703,149.129
C09936=1185.198,-47.301,-42.400,179.602,5.702,149.128
C09937=1185.192,-47.051,-42.412,179.604,5.703,149.128
C09938=1185.188,-46.802,-42.424,179.607,5.703,149.127
C09939=1185.182,-46.552,-42.435,179.609,5.704,149.127
C09940=1185.177,-46.303,-42.448,179.611,5.704,149.126
C09941=1185.171,-46.053,-42.460,179.614,5.704,149.125
C09942=1185.166,-45.803,-42.471,179.616,5.705,149.125
C09943=1185.161,-45.553,-42.483,179.619,5.705,149.124
C09944=1185.156,-45.304,-42.495,179.621,5.705,149.123
C09945=1185.151,-45.055,-42.507,179.623,5.706,149.123
C09946=1185.146,-44.805,-42.519,179.626,5.706,149.122
C09947=1185.140,-44.555,-42.530,179.628,5.707,149.121
C09948=1185.136,-44.305,-42.542,179.630,5.706,149.121
C09949=1185.131,-44.056,-42.554,179.633,5.707,149.120
C09950=1185.125,-43.806,-42.566,179.635,5.708,149.119
C09951=1185.120,-43.556,-42.578,179.638,5.708,149.119
C09952=1185.115,-43.306,-42.589,179.640,5.708,149.118
C09953=1185.110,-43.057,-42.602,179.642,5.709,149.118
C09954=1185.104,-42.807,-42.614,179.645,5.709,149.117
C09955=1185.099,-42.557,-42.626,179.647,5.709,149.116
C09956=1185.094,-42.307,-42.637,179.650,5.709,149.115
C09957=1185.089,-42.058,-42.650,179.652,5.710,149.115
C09958=1185.084,-41.808,-42.661,179.654,5.710,149.114
C09959=1185.078,-41.558,-42.673,179.657,5.711,149.114
C09960=1185.073,-41.309,-42.686,179.659,5.711,149.113
C09961=1185.069,-41.059,-42.697,179.661,5.711,149.112
C09962=1185.063,-40.809,-42.709,179.664,5.712,149.112
C09963=1185.058,-40.560,-42.722,179.667,5.712,149.111
C09964=1185.053,-40.310,-42.734,179.669,5.713,149.111
C09965=1185.047,-40.061,-42.746,179.671,5.713,149.110
C09966=1185.043,-39.811,-42.758,179.674,5.713,149.109
C09967=1185.037,-39.561,-42.769,179.676,5.714,149.109
C09968=1185.032,-39.312,-42.782,179.678,5.714,149.108
C09969=1185.027,-39.062,-42.794,179.680,5.714,149.107
C09970=1185.021,-38.812,-42.806,179.683,5.714,149.107
C09971=1185.016,-38.563,-42.818,179.685,5.715,149.106
C09972=1185.011,-38.313,-42.830,179.688,5.716,149.105
C09973=1185.006,-38.064,-42.842,179.691,5.716,149.105
C09974=1185.001,-37.814,-42.854,179.692,5.716,149.104
C09975=1184.996,-37.564,-42.867,179.695,5.717,149.104
C09976=1184.990,-37.315,-42.879,179.698,5.717,149.103
C09977=1184.985,-37.065,-42.891,179.700,5.717,149.102
C09978=1184.980,-36.815,-42.903,179.702,5.717,149.102
C09979=1184.974,-36.565,-42.915,179.704,5.718,149.101
C09980=1184.969,-36.316,-42.928,179.707,5.718,149.100
C09981=1184.965,-36.066,-42.939,179.710,5.719,149.100
C09982=1184.959,-35.817,-42.952,179.712,5.720,149.099
C09983=1184.954,-35.567,-42.963,179.714,5.719,149.098
C09984=1184.949,-35.318,-42.976,179.717,5.720,149.098
C09985=1184.943,-35.068,-42.988,179.719,5.721,149.097
C09986=1184.938,-34.819,-43.000,179.722,5.721,149.097
C09987=1184.934,-34.568,-43.013,179.724,5.721,149.096
C09988=1184.928,-34.319,-43.025,179.726,5.721,149.095
C09989=1184.923,-34.069,-43.038,179.728,5.722,149.095
C09990=1184.918,-33.819,-43.050,179.731,5.722,149.094
C09991=1184.913,-33.570,-43.062,179.734,5.723,149.093
C09992=1184.907,-33.320,-43.074,179.736,5.723,149.093
C09993=1184.902,-33.071,-43.087,179.738,5.723,149.092
C09994=1184.897,-32.821,-43.099,179.741,5.724,149.091
C09995=1184.892,-32.572,-43.111,179.743,5.724,149.091
C09996=1184.886,-32.322,-43.124,179.746,5.725,149.090
//INST
///DATE 2021/06/25 14:29
///ATTR SC,RW,RJ
////FRAME ROBOT
///GROUP1 RB1
NOP
MOVL C00000 V=800.0 PL=0
MOVL C00001 V=800.0 PL=0
MOVL C00002 V=800.0 PL=0
MOVL C00003 V=800.0 PL=0
MOVL C00004 V=800.0 PL=0
MOVL C00005 V=800.0 PL=0
MOVL C00006 V=800.0 PL=0
MOVL C00007 V=800.0 PL=0
MOVL C00008 V=800.0 PL=0
MOVL C00009 V=800.0 PL=0
MOVL C00010 V=800.0 PL=0
MOVL C00011 V=800.0 PL=0
MOVL C00012 V=800.0 PL=0
MOVL C00013 V=800.0 PL=0
MOVL C00014 V=800.0 PL=0
MOVL C00015 V=800.0 PL=0
MOVL C00016 V=800.0 PL=0
MOVL C00017 V=800.0 PL=0
MOVL C00018 V=800.0 PL=0
MOVL C00019 V=800.0 PL=0
MOVL C00020 V=800.0 PL=0
MOVL C00021 V=800.0 PL=0
MOVL C00022 V=800.0 PL=0
MOVL C00023 V=800.0 PL=0
MOVL C00024 V=800.0 PL=0
MOVL C00025 V=800.0 PL=0
MOVL C00026 V=800.0 PL=0
MOVL C00027 V=800.0 PL=0
MOVL C00028 V=800.0 PL=0
MOVL C00029 V=800.0 PL=0
MOVL C00030 V=800.0 PL=0
MOVL C00031 V=800.0 PL=0
MOVL C00032 V=800.0 PL=0
MOVL C00033 V=800.0 PL=0
MOVL C00034 V=800.0 PL=0
MOVL C00035 V=800.0 PL=0
MOVL C00036 V=800.0 PL=0
MOVL C00037 V=800.0 PL=0
MOVL C00038 V=800.0 PL=0
MOVL C00039 V=800.0 PL=0
MOVL C00040 V=800.0 PL=0
MOVL C00041 V=800.0 PL=0
MOVL C00042 V=800.0 PL=0
MOVL C00043 V=800.0 PL=0
MOVL C00044 V=800.0 PL=0
MOVL C00045 V=800.0 PL=0
MOVL C00046 V=800.0 PL=0
MOVL C00047 V=800.0 PL=0
MOVL C00048 V=800.0 PL=0
MOVL C00049 V=800.0 PL=0
MOVL C00050 V=800.0 PL=0
MOVL C00051 V=800.0 PL=0
MOVL C00052 V=800.0 PL=0
MOVL C00053 V=800.0 PL=0
MOVL C00054 V=800.0 PL=0
MOVL C00055 V=800.0 PL=0
MOVL C00056 V=800.0 PL=0
MOVL C00057 V=800.0 PL=0
MOVL C00058 V=800.0 PL=0
MOVL C00059 V=800.0 PL=0
MOVL C00060 V=800.0 PL=0
MOVL C00061 V=800.0 PL=0
MOVL C00062 V=800.0 PL=0
MOVL C00063 V=800.0 PL=0
MOVL C00064 V=800.0 PL=0
MOVL C00065 V=800.0 PL=0
MOVL C00066 V=800.0 PL=0
MOVL C00067 V=800.0 PL=0
MOVL C00068 V=800.0 PL=0
MOVL C00069 V=800.0 PL=0
MOVL C00070 V=800.0 PL=0
MOVL C00071 V=800.0 PL=0
MOVL C00072 V=800.0 PL=0
MOVL C00073 V=800.0 PL=0
MOVL C00074 V=800.0 PL=0
MOVL C00075 V=800.0 PL=0
MOVL C00076 V=800.0 PL=0
MOVL C00077 V=800.0 PL=0
MOVL C00078 V=800.0 PL=0
MOVL C00079 V=800.0 PL=0
MOVL C00080 V=800.0 PL=0
MOVL C00081 V=800.0 PL=0
MOVL C00082 V=800.0 PL=0
MOVL C00083 V=800.0 PL=0
MOVL C00084 V=800.0 PL=0
MOVL C00085 V=800.0 PL=0
MOVL C00086 V=800.0 PL=0
MOVL C00087 V=800.0 PL=0
MOVL C00088 V=800.0 PL=0
MOVL C00089 V=800.0 PL=0
MOVL C00090 V=800.0 PL=0
MOVL C00091 V=800.0 PL=0
MOVL C00092 V=800.0 PL=0
MOVL C00093 V=800.0 PL=0
MOVL C00094 V=800.0 PL=0
MOVL C00095 V=800.0 PL=0
MOVL C00096 V=800.0 PL=0
MOVL C00097 V=800.0 PL=0
MOVL C00098 V=800.0 PL=0
MOVL C00099 V=800.0 PL=0
MOVL C00100 V=800.0 PL=0
MOVL C00101 V=800.0 PL=0
MOVL C00102 V=800.0 PL=0
MOVL C00103 V=800.0 PL=0
MOVL C00104 V=800.0 PL=0
MOVL C00105 V=800.0 PL=0
MOVL C00106 V=800.0 PL=0
MOVL C00107 V=800.0 PL=0
MOVL C00108 V=800.0 PL=0
MOVL C00109 V=800.0 PL=0
MOVL C00110 V=800.0 PL=0
MOVL C00111 V=800.0 PL=0
MOVL C00112 V=800.0 PL=0
MOVL C00113 V=800.0 PL=0
MOVL C00114 V=800.0 PL=0
MOVL C00115 V=800.0 PL=0
MOVL C00116 V=800.0 PL=0
MOVL C00117 V=800.0 PL=0
MOVL C00118 V=800.0 PL=0
MOVL C00119 V=800.0 PL=0
MOVL C00120 V=800.0 PL=0
MOVL C00121 V=800.0 PL=0
MOVL C00122 V=800.0 PL=0
MOVL C00123 V=800.0 PL=0
MOVL C00124 V=800.0 PL=0
MOVL C00125 V=800.0 PL=0
MOVL C00126 V=800.0 PL=0
MOVL C00127 V=800.0 PL=0
MOVL C00128 V=800.0 PL=0
MOVL C00129 V=800.0 PL=0
MOVL C00130 V=800.0 PL=0
MOVL C00131 V=800.0 PL=0
MOVL C00132 V=800.0 PL=0
MOVL C00133 V=800.0 PL=0
MOVL C00134 V=800.0 PL=0
MOVL C00135 V=800.0 PL=0
MOVL C00136 V=800.0 PL=0
MOVL C00137 V=800.0 PL=0
MOVL C00138 V=800.0 PL=0
MOVL C00139 V=800.0 PL=0
MOVL C00140 V=800.0 PL=0
MOVL C00141 V=800.0 PL=0
MOVL C00142 V=800.0 PL=0
MOVL C00143 V=800.0 PL=0
MOVL C00144 V=800.0 PL=0
MOVL C00145 V=800.0 PL=0
MOVL C00146 V=800.0 PL=0
MOVL C00147 V=800.0 PL=0
MOVL C00148 V=800.0 PL=0
MOVL C00149 V=800.0 PL=0
MOVL C00150 V=800.0 PL=0
MOVL C00151 V=800.0 PL=0
MOVL C00152 V=800.0 PL=0
MOVL C00153 V=800.0 PL=0
MOVL C00154 V=800.0 PL=0
MOVL C00155 V=800.0 PL=0
MOVL C00156 V=800.0 PL=0
MOVL C00157 V=800.0 PL=0
MOVL C00158 V=800.0 PL=0
MOVL C00159 V=800.0 PL=0
MOVL C00160 V=800.0 PL=0
MOVL C00161 V=800.0 PL=0
MOVL C00162 V=800.0 PL=0
MOVL C00163 V=800.0 PL=0
MOVL C00164 V=800.0 PL=0
MOVL C00165 V=800.0 PL=0
MOVL C00166 V=800.0 PL=0
MOVL C00167 V=800.0 PL=0
MOVL C00168 V=800.0 PL=0
MOVL C00169 V=800.0 PL=0
MOVL C00170 V=800.0 PL=0
MOVL C00171 V=800.0 PL=0
MOVL C00172 V=800.0 PL=0
MOVL C00173 V=800.0 PL=0
MOVL C00174 V=800.0 PL=0
MOVL C00175 V=800.0 PL=0
MOVL C00176 V=800.0 PL=0
MOVL C00177 V=800.0 PL=0
MOVL C00178 V=800.0 PL=0
MOVL C00179 V=800.0 PL=0
MOVL C00180 V=800.0 PL=0
MOVL C00181 V=800.0 PL=0
MOVL C00182 V=800.0 PL=0
MOVL C00183 V=800.0 PL=0
MOVL C00184 V=800.0 PL=0
MOVL C00185 V=800.0 PL=0
MOVL C00186 V=800.0 PL=0
MOVL C00187 V=800.0 PL=0
MOVL C00188 V=800.0 PL=0
MOVL C00189 V=800.0 PL=0
MOVL C00190 V=800.0 PL=0
MOVL C00191 V=800.0 PL=0
MOVL C00192 V=800.0 PL=0
MOVL C00193 V=800.0 PL=0
MOVL C00194 V=800.0 PL=0
MOVL C00195 V=800.0 PL=0
MOVL C00196 V=800.0 PL=0
MOVL C00197 V=800.0 PL=0
MOVL C00198 V=800.0 PL=0
MOVL C00199 V=800.0 PL=0
MOVL C00200 V=800.0 PL=0
MOVL C00201 V=800.0 PL=0
MOVL C00202 V=800.0 PL=0
MOVL C00203 V=800.0 PL=0
MOVL C00204 V=800.0 PL=0
MOVL C00205 V=800.0 PL=0
MOVL C00206 V=800.0 PL=0
MOVL C00207 V=800.0 PL=0
MOVL C00208 V=800.0 PL=0
MOVL C00209 V=800.0 PL=0
MOVL C00210 V=800.0 PL=0
MOVL C00211 V=800.0 PL=0
MOVL C00212 V=800.0 PL=0
MOVL C00213 V=800.0 PL=0
MOVL C00214 V=800.0 PL=0
MOVL C00215 V=800.0 PL=0
MOVL C00216 V=800.0 PL=0
MOVL C00217 V=800.0 PL=0
MOVL C00218 V=800.0 PL=0
MOVL C00219 V=800.0 PL=0
MOVL C00220 V=800.0 PL=0
MOVL C00221 V=800.0 PL=0
MOVL C00222 V=800.0 PL=0
MOVL C00223 V=800.0 PL=0
MOVL C00224 V=800.0 PL=0
MOVL C00225 V=800.0 PL=0
MOVL C00226 V=800.0 PL=0
MOVL C00227 V=800.0 PL=0
MOVL C00228 V=800.0 PL=0
MOVL C00229 V=800.0 PL=0
MOVL C00230 V=800.0 PL=0
MOVL C00231 V=800.0 PL=0
MOVL C00232 V=800.0 PL=0
MOVL C00233 V=800.0 PL=0
MOVL C00234 V=800.0 PL=0
MOVL C00235 V=800.0 PL=0
MOVL C00236 V=800.0 PL=0
MOVL C00237 V=800.0 PL=0
MOVL C00238 V=800.0 PL=0
MOVL C00239 V=800.0 PL=0
MOVL C00240 V=800.0 PL=0
MOVL C00241 V=800.0 PL=0
MOVL C00242 V=800.0 PL=0
MOVL C00243 V=800.0 PL=0
MOVL C00244 V=800.0 PL=0
MOVL C00245 V=800.0 PL=0
MOVL C00246 V=800.0 PL=0
MOVL C00247 V=800.0 PL=0
MOVL C00248 V=800.0 PL=0
MOVL C00249 V=800.0 PL=0
MOVL C00250 V=800.0 PL=0
MOVL C00251 V=800.0 PL=0
MOVL C00252 V=800.0 PL=0
MOVL C00253 V=800.0 PL=0
MOVL C00254 V=800.0 PL=0
MOVL C00255 V=800.0 PL=0
MOVL C00256 V=800.0 PL=0
MOVL C00257 V=800.0 PL=0
MOVL C00258 V=800.0 PL=0
MOVL C00259 V=800.0 PL=0
MOVL C00260 V=800.0 PL=0
MOVL C00261 V=800.0 PL=0
MOVL C00262 V=800.0 PL=0
MOVL C00263 V=800.0 PL=0
MOVL C00264 V=800.0 PL=0
MOVL C00265 V=800.0 PL=0
MOVL C00266 V=800.0 PL=0
MOVL C00267 V=800.0 PL=0
MOVL C00268 V=800.0 PL=0
MOVL C00269 V=800.0 PL=0
MOVL C00270 V=800.0 PL=0
MOVL C00271 V=800.0 PL=0
MOVL C00272 V=800.0 PL=0
MOVL C00273 V=800.0 PL=0
MOVL C00274 V=800.0 PL=0
MOVL C00275 V=800.0 PL=0
MOVL C00276 V=800.0 PL=0
MOVL C00277 V=800.0 PL=0
MOVL C00278 V=800.0 PL=0
MOVL C00279 V=800.0 PL=0
MOVL C00280 V=800.0 PL=0
MOVL C00281 V=800.0 PL=0
MOVL C00282 V=800.0 PL=0
MOVL C00283 V=800.0 PL=0
MOVL C00284 V=800.0 PL=0
MOVL C00285 V=800.0 PL=0
MOVL C00286 V=800.0 PL=0
MOVL C00287 V=800.0 PL=0
MOVL C00288 V=800.0 PL=0
MOVL C00289 V=800.0 PL=0
MOVL C00290 V=800.0 PL=0
MOVL C00291 V=800.0 PL=0
MOVL C00292 V=800.0 PL=0
MOVL C00293 V=800.0 PL=0
MOVL C00294 V=800.0 PL=0
MOVL C00295 V=800.0 PL=0
MOVL C00296 V=800.0 PL=0
MOVL C00297 V=800.0 PL=0
MOVL C00298 V=800.0 PL=0
MOVL C00299 V=800.0 PL=0
MOVL C00300 V=800.0 PL=0
MOVL C00301 V=800.0 PL=0
MOVL C00302 V=800.0 PL=0
MOVL C00303 V=800.0 PL=0
MOVL C00304 V=800.0 PL=0
MOVL C00305 V=800.0 PL=0
MOVL C00306 V=800.0 PL=0
MOVL C00307 V=800.0 PL=0
MOVL C00308 V=800.0 PL=0
MOVL C00309 V=800.0 PL=0
MOVL C00310 V=800.0 PL=0
MOVL C00311 V=800.0 PL=0
MOVL C00312 V=800.0 PL=0
MOVL C00313 V=800.0 PL=0
MOVL C00314 V=800.0 PL=0
MOVL C00315 V=800.0 PL=0
MOVL C00316 V=800.0 PL=0
MOVL C00317 V=800.0 PL=0
MOVL C00318 V=800.0 PL=0
MOVL C00319 V=800.0 PL=0
MOVL C00320 V=800.0 PL=0
MOVL C00321 V=800.0 PL=0
MOVL C00322 V=800.0 PL=0
MOVL C00323 V=800.0 PL=0
MOVL C00324 V=800.0 PL=0
MOVL C00325 V=800.0 PL=0
MOVL C00326 V=800.0 PL=0
MOVL C00327 V=800.0 PL=0
MOVL C00328 V=800.0 PL=0
MOVL C00329 V=800.0 PL=0
MOVL C00330 V=800.0 PL=0
MOVL C00331 V=800.0 PL=0
MOVL C00332 V=800.0 PL=0
MOVL C00333 V=800.0 PL=0
MOVL C00334 V=800.0 PL=0
MOVL C00335 V=800.0 PL=0
MOVL C00336 V=800.0 PL=0
MOVL C00337 V=800.0 PL=0
MOVL C00338 V=800.0 PL=0
MOVL C00339 V=800.0 PL=0
MOVL C00340 V=800.0 PL=0
MOVL C00341 V=800.0 PL=0
MOVL C00342 V=800.0 PL=0
MOVL C00343 V=800.0 PL=0
MOVL C00344 V=800.0 PL=0
MOVL C00345 V=800.0 PL=0
MOVL C00346 V=800.0 PL=0
MOVL C00347 V=800.0 PL=0
MOVL C00348 V=800.0 PL=0
MOVL C00349 V=800.0 PL=0
MOVL C00350 V=800.0 PL=0
MOVL C00351 V=800.0 PL=0
MOVL C00352 V=800.0 PL=0
MOVL C00353 V=800.0 PL=0
MOVL C00354 V=800.0 PL=0
MOVL C00355 V=800.0 PL=0
MOVL C00356 V=800.0 PL=0
MOVL C00357 V=800.0 PL=0
MOVL C00358 V=800.0 PL=0
MOVL C00359 V=800.0 PL=0
MOVL C00360 V=800.0 PL=0
MOVL C00361 V=800.0 PL=0
MOVL C00362 V=800.0 PL=0
MOVL C00363 V=800.0 PL=0
MOVL C00364 V=800.0 PL=0
MOVL C00365 V=800.0 PL=0
MOVL C00366 V=800.0 PL=0
MOVL C00367 V=800.0 PL=0
MOVL C00368 V=800.0 PL=0
MOVL C00369 V=800.0 PL=0
MOVL C00370 V=800.0 PL=0
MOVL C00371 V=800.0 PL=0
MOVL C00372 V=800.0 PL=0
MOVL C00373 V=800.0 PL=0
MOVL C00374 V=800.0 PL=0
MOVL C00375 V=800.0 PL=0
MOVL C00376 V=800.0 PL=0
MOVL C00377 V=800.0 PL=0
MOVL C00378 V=800.0 PL=0
MOVL C00379 V=800.0 PL=0
MOVL C00380 V=800.0 PL=0
MOVL C00381 V=800.0 PL=0
MOVL C00382 V=800.0 PL=0
MOVL C00383 V=800.0 PL=0
MOVL C00384 V=800.0 PL=0
MOVL C00385 V=800.0 PL=0
MOVL C00386 V=800.0 PL=0
MOVL C00387 V=800.0 PL=0
MOVL C00388 V=800.0 PL=0
MOVL C00389 V=800.0 PL=0
MOVL C00390 V=800.0 PL=0
MOVL C00391 V=800.0 PL=0
MOVL C00392 V=800.0 PL=0
MOVL C00393 V=800.0 PL=0
MOVL C00394 V=800.0 PL=0
MOVL C00395 V=800.0 PL=0
MOVL C00396 V=800.0 PL=0
MOVL C00397 V=800.0 PL=0
MOVL C00398 V=800.0 PL=0
MOVL C00399 V=800.0 PL=0
MOVL C00400 V=800.0 PL=0
MOVL C00401 V=800.0 PL=0
MOVL C00402 V=800.0 PL=0
MOVL C00403 V=800.0 PL=0
MOVL C00404 V=800.0 PL=0
MOVL C00405 V=800.0 PL=0
MOVL C00406 V=800.0 PL=0
MOVL C00407 V=800.0 PL=0
MOVL C00408 V=800.0 PL=0
MOVL C00409 V=800.0 PL=0
MOVL C00410 V=800.0 PL=0
MOVL C00411 V=800.0 PL=0
MOVL C00412 V=800.0 PL=0
MOVL C00413 V=800.0 PL=0
MOVL C00414 V=800.0 PL=0
MOVL C00415 V=800.0 PL=0
MOVL C00416 V=800.0 PL=0
MOVL C00417 V=800.0 PL=0
MOVL C00418 V=800.0 PL=0
MOVL C00419 V=800.0 PL=0
MOVL C00420 V=800.0 PL=0
MOVL C00421 V=800.0 PL=0
MOVL C00422 V=800.0 PL=0
MOVL C00423 V=800.0 PL=0
MOVL C00424 V=800.0 PL=0
MOVL C00425 V=800.0 PL=0
MOVL C00426 V=800.0 PL=0
MOVL C00427 V=800.0 PL=0
MOVL C00428 V=800.0 PL=0
MOVL C00429 V=800.0 PL=0
MOVL C00430 V=800.0 PL=0
MOVL C00431 V=800.0 PL=0
MOVL C00432 V=800.0 PL=0
MOVL C00433 V=800.0 PL=0
MOVL C00434 V=800.0 PL=0
MOVL C00435 V=800.0 PL=0
MOVL C00436 V=800.0 PL=0
MOVL C00437 V=800.0 PL=0
MOVL C00438 V=800.0 PL=0
MOVL C00439 V=800.0 PL=0
MOVL C00440 V=800.0 PL=0
MOVL C00441 V=800.0 PL=0
MOVL C00442 V=800.0 PL=0
MOVL C00443 V=800.0 PL=0
MOVL C00444 V=800.0 PL=0
MOVL C00445 V=800.0 PL=0
MOVL C00446 V=800.0 PL=0
MOVL C00447 V=800.0 PL=0
MOVL C00448 V=800.0 PL=0
MOVL C00449 V=800.0 PL=0
MOVL C00450 V=800.0 PL=0
MOVL C00451 V=800.0 PL=0
MOVL C00452 V=800.0 PL=0
MOVL C00453 V=800.0 PL=0
MOVL C00454 V=800.0 PL=0
MOVL C00455 V=800.0 PL=0
MOVL C00456 V=800.0 PL=0
MOVL C00457 V=800.0 PL=0
MOVL C00458 V=800.0 PL=0
MOVL C00459 V=800.0 PL=0
MOVL C00460 V=800.0 PL=0
MOVL C00461 V=800.0 PL=0
MOVL C00462 V=800.0 PL=0
MOVL C00463 V=800.0 PL=0
MOVL C00464 V=800.0 PL=0
MOVL C00465 V=800.0 PL=0
MOVL C00466 V=800.0 PL=0
MOVL C00467 V=800.0 PL=0
MOVL C00468 V=800.0 PL=0
MOVL C00469 V=800.0 PL=0
MOVL C00470 V=800.0 PL=0
MOVL C00471 V=800.0 PL=0
MOVL C00472 V=800.0 PL=0
MOVL C00473 V=800.0 PL=0
MOVL C00474 V=800.0 PL=0
MOVL C00475 V=800.0 PL=0
MOVL C00476 V=800.0 PL=0
MOVL C00477 V=800.0 PL=0
MOVL C00478 V=800.0 PL=0
MOVL C00479 V=800.0 PL=0
MOVL C00480 V=800.0 PL=0
MOVL C00481 V=800.0 PL=0
MOVL C00482 V=800.0 PL=0
MOVL C00483 V=800.0 PL=0
MOVL C00484 V=800.0 PL=0
MOVL C00485 V=800.0 PL=0
MOVL C00486 V=800.0 PL=0
MOVL C00487 V=800.0 PL=0
MOVL C00488 V=800.0 PL=0
MOVL C00489 V=800.0 PL=0
MOVL C00490 V=800.0 PL=0
MOVL C00491 V=800.0 PL=0
MOVL C00492 V=800.0 PL=0
MOVL C00493 V=800.0 PL=0
MOVL C00494 V=800.0 PL=0
MOVL C00495 V=800.0 PL=0
MOVL C00496 V=800.0 PL=0
MOVL C00497 V=800.0 PL=0
MOVL C00498 V=800.0 PL=0
MOVL C00499 V=800.0 PL=0
MOVL C00500 V=800.0 PL=0
MOVL C00501 V=800.0 PL=0
MOVL C00502 V=800.0 PL=0
MOVL C00503 V=800.0 PL=0
MOVL C00504 V=800.0 PL=0
MOVL C00505 V=800.0 PL=0
MOVL C00506 V=800.0 PL=0
MOVL C00507 V=800.0 PL=0
MOVL C00508 V=800.0 PL=0
MOVL C00509 V=800.0 PL=0
MOVL C00510 V=800.0 PL=0
MOVL C00511 V=800.0 PL=0
MOVL C00512 V=800.0 PL=0
MOVL C00513 V=800.0 PL=0
MOVL C00514 V=800.0 PL=0
MOVL C00515 V=800.0 PL=0
MOVL C00516 V=800.0 PL=0
MOVL C00517 V=800.0 PL=0
MOVL C00518 V=800.0 PL=0
MOVL C00519 V=800.0 PL=0
MOVL C00520 V=800.0 PL=0
MOVL C00521 V=800.0 PL=0
MOVL C00522 V=800.0 PL=0
MOVL C00523 V=800.0 PL=0
MOVL C00524 V=800.0 PL=0
MOVL C00525 V=800.0 PL=0
MOVL C00526 V=800.0 PL=0
MOVL C00527 V=800.0 PL=0
MOVL C00528 V=800.0 PL=0
MOVL C00529 V=800.0 PL=0
MOVL C00530 V=800.0 PL=0
MOVL C00531 V=800.0 PL=0
MOVL C00532 V=800.0 PL=0
MOVL C00533 V=800.0 PL=0
MOVL C00534 V=800.0 PL=0
MOVL C00535 V=800.0 PL=0
MOVL C00536 V=800.0 PL=0
MOVL C00537 V=800.0 PL=0
MOVL C00538 V=800.0 PL=0
MOVL C00539 V=800.0 PL=0
MOVL C00540 V=800.0 PL=0
MOVL C00541 V=800.0 PL=0
MOVL C00542 V=800.0 PL=0
MOVL C00543 V=800.0 PL=0
MOVL C00544 V=800.0 PL=0
MOVL C00545 V=800.0 PL=0
MOVL C00546 V=800.0 PL=0
MOVL C00547 V=800.0 PL=0
MOVL C00548 V=800.0 PL=0
MOVL C00549 V=800.0 PL=0
MOVL C00550 V=800.0 PL=0
MOVL C00551 V=800.0 PL=0
MOVL C00552 V=800.0 PL=0
MOVL C00553 V=800.0 PL=0
MOVL C00554 V=800.0 PL=0
MOVL C00555 V=800.0 PL=0
MOVL C00556 V=800.0 PL=0
MOVL C00557 V=800.0 PL=0
MOVL C00558 V=800.0 PL=0
MOVL C00559 V=800.0 PL=0
MOVL C00560 V=800.0 PL=0
MOVL C00561 V=800.0 PL=0
MOVL C00562 V=800.0 PL=0
MOVL C00563 V=800.0 PL=0
MOVL C00564 V=800.0 PL=0
MOVL C00565 V=800.0 PL=0
MOVL C00566 V=800.0 PL=0
MOVL C00567 V=800.0 PL=0
MOVL C00568 V=800.0 PL=0
MOVL C00569 V=800.0 PL=0
MOVL C00570 V=800.0 PL=0
MOVL C00571 V=800.0 PL=0
MOVL C00572 V=800.0 PL=0
MOVL C00573 V=800.0 PL=0
MOVL C00574 V=800.0 PL=0
MOVL C00575 V=800.0 PL=0
MOVL C00576 V=800.0 PL=0
MOVL C00577 V=800.0 PL=0
MOVL C00578 V=800.0 PL=0
MOVL C00579 V=800.0 PL=0
MOVL C00580 V=800.0 PL=0
MOVL C00581 V=800.0 PL=0
MOVL C00582 V=800.0 PL=0
MOVL C00583 V=800.0 PL=0
MOVL C00584 V=800.0 PL=0
MOVL C00585 V=800.0 PL=0
MOVL C00586 V=800.0 PL=0
MOVL C00587 V=800.0 PL=0
MOVL C00588 V=800.0 PL=0
MOVL C00589 V=800.0 PL=0
MOVL C00590 V=800.0 PL=0
MOVL C00591 V=800.0 PL=0
MOVL C00592 V=800.0 PL=0
MOVL C00593 V=800.0 PL=0
MOVL C00594 V=800.0 PL=0
MOVL C00595 V=800.0 PL=0
MOVL C00596 V=800.0 PL=0
MOVL C00597 V=800.0 PL=0
MOVL C00598 V=800.0 PL=0
MOVL C00599 V=800.0 PL=0
MOVL C00600 V=800.0 PL=0
MOVL C00601 V=800.0 PL=0
MOVL C00602 V=800.0 PL=0
MOVL C00603 V=800.0 PL=0
MOVL C00604 V=800.0 PL=0
MOVL C00605 V=800.0 PL=0
MOVL C00606 V=800.0 PL=0
MOVL C00607 V=800.0 PL=0
MOVL C00608 V=800.0 PL=0
MOVL C00609 V=800.0 PL=0
MOVL C00610 V=800.0 PL=0
MOVL C00611 V=800.0 PL=0
MOVL C00612 V=800.0 PL=0
MOVL C00613 V=800.0 PL=0
MOVL C00614 V=800.0 PL=0
MOVL C00615 V=800.0 PL=0
MOVL C00616 V=800.0 PL=0
MOVL C00617 V=800.0 PL=0
MOVL C00618 V=800.0 PL=0
MOVL C00619 V=800.0 PL=0
MOVL C00620 V=800.0 PL=0
MOVL C00621 V=800.0 PL=0
MOVL C00622 V=800.0 PL=0
MOVL C00623 V=800.0 PL=0
MOVL C00624 V=800.0 PL=0
MOVL C00625 V=800.0 PL=0
MOVL C00626 V=800.0 PL=0
MOVL C00627 V=800.0 PL=0
MOVL C00628 V=800.0 PL=0
MOVL C00629 V=800.0 PL=0
MOVL C00630 V=800.0 PL=0
MOVL C00631 V=800.0 PL=0
MOVL C00632 V=800.0 PL=0
MOVL C00633 V=800.0 PL=0
MOVL C00634 V=800.0 PL=0
MOVL C00635 V=800.0 PL=0
MOVL C00636 V=800.0 PL=0
MOVL C00637 V=800.0 PL=0
MOVL C00638 V=800.0 PL=0
MOVL C00639 V=800.0 PL=0
MOVL C00640 V=800.0 PL=0
MOVL C00641 V=800.0 PL=0
MOVL C00642 V=800.0 PL=0
MOVL C00643 V=800.0 PL=0
MOVL C00644 V=800.0 PL=0
MOVL C00645 V=800.0 PL=0
MOVL C00646 V=800.0 PL=0
MOVL C00647 V=800.0 PL=0
MOVL C00648 V=800.0 PL=0
MOVL C00649 V=800.0 PL=0
MOVL C00650 V=800.0 PL=0
MOVL C00651 V=800.0 PL=0
MOVL C00652 V=800.0 PL=0
MOVL C00653 V=800.0 PL=0
MOVL C00654 V=800.0 PL=0
MOVL C00655 V=800.0 PL=0
MOVL C00656 V=800.0 PL=0
MOVL C00657 V=800.0 PL=0
MOVL C00658 V=800.0 PL=0
MOVL C00659 V=800.0 PL=0
MOVL C00660 V=800.0 PL=0
MOVL C00661 V=800.0 PL=0
MOVL C00662 V=800.0 PL=0
MOVL C00663 V=800.0 PL=0
MOVL C00664 V=800.0 PL=0
MOVL C00665 V=800.0 PL=0
MOVL C00666 V=800.0 PL=0
MOVL C00667 V=800.0 PL=0
MOVL C00668 V=800.0 PL=0
MOVL C00669 V=800.0 PL=0
MOVL C00670 V=800.0 PL=0
MOVL C00671 V=800.0 PL=0
MOVL C00672 V=800.0 PL=0
MOVL C00673 V=800.0 PL=0
MOVL C00674 V=800.0 PL=0
MOVL C00675 V=800.0 PL=0
MOVL C00676 V=800.0 PL=0
MOVL C00677 V=800.0 PL=0
MOVL C00678 V=800.0 PL=0
MOVL C00679 V=800.0 PL=0
MOVL C00680 V=800.0 PL=0
MOVL C00681 V=800.0 PL=0
MOVL C00682 V=800.0 PL=0
MOVL C00683 V=800.0 PL=0
MOVL C00684 V=800.0 PL=0
MOVL C00685 V=800.0 PL=0
MOVL C00686 V=800.0 PL=0
MOVL C00687 V=800.0 PL=0
MOVL C00688 V=800.0 PL=0
MOVL C00689 V=800.0 PL=0
MOVL C00690 V=800.0 PL=0
MOVL C00691 V=800.0 PL=0
MOVL C00692 V=800.0 PL=0
MOVL C00693 V=800.0 PL=0
MOVL C00694 V=800.0 PL=0
MOVL C00695 V=800.0 PL=0
MOVL C00696 V=800.0 PL=0
MOVL C00697 V=800.0 PL=0
MOVL C00698 V=800.0 PL=0
MOVL C00699 V=800.0 PL=0
MOVL C00700 V=800.0 PL=0
MOVL C00701 V=800.0 PL=0
MOVL C00702 V=800.0 PL=0
MOVL C00703 V=800.0 PL=0
MOVL C00704 V=800.0 PL=0
MOVL C00705 V=800.0 PL=0
MOVL C00706 V=800.0 PL=0
MOVL C00707 V=800.0 PL=0
MOVL C00708 V=800.0 PL=0
MOVL C00709 V=800.0 PL=0
MOVL C00710 V=800.0 PL=0
MOVL C00711 V=800.0 PL=0
MOVL C00712 V=800.0 PL=0
MOVL C00713 V=800.0 PL=0
MOVL C00714 V=800.0 PL=0
MOVL C00715 V=800.0 PL=0
MOVL C00716 V=800.0 PL=0
MOVL C00717 V=800.0 PL=0
MOVL C00718 V=800.0 PL=0
MOVL C00719 V=800.0 PL=0
MOVL C00720 V=800.0 PL=0
MOVL C00721 V=800.0 PL=0
MOVL C00722 V=800.0 PL=0
MOVL C00723 V=800.0 PL=0
MOVL C00724 V=800.0 PL=0
MOVL C00725 V=800.0 PL=0
MOVL C00726 V=800.0 PL=0
MOVL C00727 V=800.0 PL=0
MOVL C00728 V=800.0 PL=0
MOVL C00729 V=800.0 PL=0
MOVL C00730 V=800.0 PL=0
MOVL C00731 V=800.0 PL=0
MOVL C00732 V=800.0 PL=0
MOVL C00733 V=800.0 PL=0
MOVL C00734 V=800.0 PL=0
MOVL C00735 V=800.0 PL=0
MOVL C00736 V=800.0 PL=0
MOVL C00737 V=800.0 PL=0
MOVL C00738 V=800.0 PL=0
MOVL C00739 V=800.0 PL=0
MOVL C00740 V=800.0 PL=0
MOVL C00741 V=800.0 PL=0
MOVL C00742 V=800.0 PL=0
MOVL C00743 V=800.0 PL=0
MOVL C00744 V=800.0 PL=0
MOVL C00745 V=800.0 PL=0
MOVL C00746 V=800.0 PL=0
MOVL C00747 V=800.0 PL=0
MOVL C00748 V=800.0 PL=0
MOVL C00749 V=800.0 PL=0
MOVL C00750 V=800.0 PL=0
MOVL C00751 V=800.0 PL=0
MOVL C00752 V=800.0 PL=0
MOVL C00753 V=800.0 PL=0
MOVL C00754 V=800.0 PL=0
MOVL C00755 V=800.0 PL=0
MOVL C00756 V=800.0 PL=0
MOVL C00757 V=800.0 PL=0
MOVL C00758 V=800.0 PL=0
MOVL C00759 V=800.0 PL=0
MOVL C00760 V=800.0 PL=0
MOVL C00761 V=800.0 PL=0
MOVL C00762 V=800.0 PL=0
MOVL C00763 V=800.0 PL=0
MOVL C00764 V=800.0 PL=0
MOVL C00765 V=800.0 PL=0
MOVL C00766 V=800.0 PL=0
MOVL C00767 V=800.0 PL=0
MOVL C00768 V=800.0 PL=0
MOVL C00769 V=800.0 PL=0
MOVL C00770 V=800.0 PL=0
MOVL C00771 V=800.0 PL=0
MOVL C00772 V=800.0 PL=0
MOVL C00773 V=800.0 PL=0
MOVL C00774 V=800.0 PL=0
MOVL C00775 V=800.0 PL=0
MOVL C00776 V=800.0 PL=0
MOVL C00777 V=800.0 PL=0
MOVL C00778 V=800.0 PL=0
MOVL C00779 V=800.0 PL=0
MOVL C00780 V=800.0 PL=0
MOVL C00781 V=800.0 PL=0
MOVL C00782 V=800.0 PL=0
MOVL C00783 V=800.0 PL=0
MOVL C00784 V=800.0 PL=0
MOVL C00785 V=800.0 PL=0
MOVL C00786 V=800.0 PL=0
MOVL C00787 V=800.0 PL=0
MOVL C00788 V=800.0 PL=0
MOVL C00789 V=800.0 PL=0
MOVL C00790 V=800.0 PL=0
MOVL C00791 V=800.0 PL=0
MOVL C00792 V=800.0 PL=0
MOVL C00793 V=800.0 PL=0
MOVL C00794 V=800.0 PL=0
MOVL C00795 V=800.0 PL=0
MOVL C00796 V=800.0 PL=0
MOVL C00797 V=800.0 PL=0
MOVL C00798 V=800.0 PL=0
MOVL C00799 V=800.0 PL=0
MOVL C00800 V=800.0 PL=0
MOVL C00801 V=800.0 PL=0
MOVL C00802 V=800.0 PL=0
MOVL C00803 V=800.0 PL=0
MOVL C00804 V=800.0 PL=0
MOVL C00805 V=800.0 PL=0
MOVL C00806 V=800.0 PL=0
MOVL C00807 V=800.0 PL=0
MOVL C00808 V=800.0 PL=0
MOVL C00809 V=800.0 PL=0
MOVL C00810 V=800.0 PL=0
MOVL C00811 V=800.0 PL=0
MOVL C00812 V=800.0 PL=0
MOVL C00813 V=800.0 PL=0
MOVL C00814 V=800.0 PL=0
MOVL C00815 V=800.0 PL=0
MOVL C00816 V=800.0 PL=0
MOVL C00817 V=800.0 PL=0
MOVL C00818 V=800.0 PL=0
MOVL C00819 V=800.0 PL=0
MOVL C00820 V=800.0 PL=0
MOVL C00821 V=800.0 PL=0
MOVL C00822 V=800.0 PL=0
MOVL C00823 V=800.0 PL=0
MOVL C00824 V=800.0 PL=0
MOVL C00825 V=800.0 PL=0
MOVL C00826 V=800.0 PL=0
MOVL C00827 V=800.0 PL=0
MOVL C00828 V=800.0 PL=0
MOVL C00829 V=800.0 PL=0
MOVL C00830 V=800.0 PL=0
MOVL C00831 V=800.0 PL=0
MOVL C00832 V=800.0 PL=0
MOVL C00833 V=800.0 PL=0
MOVL C00834 V=800.0 PL=0
MOVL C00835 V=800.0 PL=0
MOVL C00836 V=800.0 PL=0
MOVL C00837 V=800.0 PL=0
MOVL C00838 V=800.0 PL=0
MOVL C00839 V=800.0 PL=0
MOVL C00840 V=800.0 PL=0
MOVL C00841 V=800.0 PL=0
MOVL C00842 V=800.0 PL=0
MOVL C00843 V=800.0 PL=0
MOVL C00844 V=800.0 PL=0
MOVL C00845 V=800.0 PL=0
MOVL C00846 V=800.0 PL=0
MOVL C00847 V=800.0 PL=0
MOVL C00848 V=800.0 PL=0
MOVL C00849 V=800.0 PL=0
MOVL C00850 V=800.0 PL=0
MOVL C00851 V=800.0 PL=0
MOVL C00852 V=800.0 PL=0
MOVL C00853 V=800.0 PL=0
MOVL C00854 V=800.0 PL=0
MOVL C00855 V=800.0 PL=0
MOVL C00856 V=800.0 PL=0
MOVL C00857 V=800.0 PL=0
MOVL C00858 V=800.0 PL=0
MOVL C00859 V=800.0 PL=0
MOVL C00860 V=800.0 PL=0
MOVL C00861 V=800.0 PL=0
MOVL C00862 V=800.0 PL=0
MOVL C00863 V=800.0 PL=0
MOVL C00864 V=800.0 PL=0
MOVL C00865 V=800.0 PL=0
MOVL C00866 V=800.0 PL=0
MOVL C00867 V=800.0 PL=0
MOVL C00868 V=800.0 PL=0
MOVL C00869 V=800.0 PL=0
MOVL C00870 V=800.0 PL=0
MOVL C00871 V=800.0 PL=0
MOVL C00872 V=800.0 PL=0
MOVL C00873 V=800.0 PL=0
MOVL C00874 V=800.0 PL=0
MOVL C00875 V=800.0 PL=0
MOVL C00876 V=800.0 PL=0
MOVL C00877 V=800.0 PL=0
MOVL C00878 V=800.0 PL=0
MOVL C00879 V=800.0 PL=0
MOVL C00880 V=800.0 PL=0
MOVL C00881 V=800.0 PL=0
MOVL C00882 V=800.0 PL=0
MOVL C00883 V=800.0 PL=0
MOVL C00884 V=800.0 PL=0
MOVL C00885 V=800.0 PL=0
MOVL C00886 V=800.0 PL=0
MOVL C00887 V=800.0 PL=0
MOVL C00888 V=800.0 PL=0
MOVL C00889 V=800.0 PL=0
MOVL C00890 V=800.0 PL=0
MOVL C00891 V=800.0 PL=0
MOVL C00892 V=800.0 PL=0
MOVL C00893 V=800.0 PL=0
MOVL C00894 V=800.0 PL=0
MOVL C00895 V=800.0 PL=0
MOVL C00896 V=800.0 PL=0
MOVL C00897 V=800.0 PL=0
MOVL C00898 V=800.0 PL=0
MOVL C00899 V=800.0 PL=0
MOVL C00900 V=800.0 PL=0
MOVL C00901 V=800.0 PL=0
MOVL C00902 V=800.0 PL=0
MOVL C00903 V=800.0 PL=0
MOVL C00904 V=800.0 PL=0
MOVL C00905 V=800.0 PL=0
MOVL C00906 V=800.0 PL=0
MOVL C00907 V=800.0 PL=0
MOVL C00908 V=800.0 PL=0
MOVL C00909 V=800.0 PL=0
MOVL C00910 V=800.0 PL=0
MOVL C00911 V=800.0 PL=0
MOVL C00912 V=800.0 PL=0
MOVL C00913 V=800.0 PL=0
MOVL C00914 V=800.0 PL=0
MOVL C00915 V=800.0 PL=0
MOVL C00916 V=800.0 PL=0
MOVL C00917 V=800.0 PL=0
MOVL C00918 V=800.0 PL=0
MOVL C00919 V=800.0 PL=0
MOVL C00920 V=800.0 PL=0
MOVL C00921 V=800.0 PL=0
MOVL C00922 V=800.0 PL=0
MOVL C00923 V=800.0 PL=0
MOVL C00924 V=800.0 PL=0
MOVL C00925 V=800.0 PL=0
MOVL C00926 V=800.0 PL=0
MOVL C00927 V=800.0 PL=0
MOVL C00928 V=800.0 PL=0
MOVL C00929 V=800.0 PL=0
MOVL C00930 V=800.0 PL=0
MOVL C00931 V=800.0 PL=0
MOVL C00932 V=800.0 PL=0
MOVL C00933 V=800.0 PL=0
MOVL C00934 V=800.0 PL=0
MOVL C00935 V=800.0 PL=0
MOVL C00936 V=800.0 PL=0
MOVL C00937 V=800.0 PL=0
MOVL C00938 V=800.0 PL=0
MOVL C00939 V=800.0 PL=0
MOVL C00940 V=800.0 PL=0
MOVL C00941 V=800.0 PL=0
MOVL C00942 V=800.0 PL=0
MOVL C00943 V=800.0 PL=0
MOVL C00944 V=800.0 PL=0
MOVL C00945 V=800.0 PL=0
MOVL C00946 V=800.0 PL=0
MOVL C00947 V=800.0 PL=0
MOVL C00948 V=800.0 PL=0
MOVL C00949 V=800.0 PL=0
MOVL C00950 V=800.0 PL=0
MOVL C00951 V=800.0 PL=0
MOVL C00952 V=800.0 PL=0
MOVL C00953 V=800.0 PL=0
MOVL C00954 V=800.0 PL=0
MOVL C00955 V=800.0 PL=0
MOVL C00956 V=800.0 PL=0
MOVL C00957 V=800.0 PL=0
MOVL C00958 V=800.0 PL=0
MOVL C00959 V=800.0 PL=0
MOVL C00960 V=800.0 PL=0
MOVL C00961 V=800.0 PL=0
MOVL C00962 V=800.0 PL=0
MOVL C00963 V=800.0 PL=0
MOVL C00964 V=800.0 PL=0
MOVL C00965 V=800.0 PL=0
MOVL C00966 V=800.0 PL=0
MOVL C00967 V=800.0 PL=0
MOVL C00968 V=800.0 PL=0
MOVL C00969 V=800.0 PL=0
MOVL C00970 V=800.0 PL=0
MOVL C00971 V=800.0 PL=0
MOVL C00972 V=800.0 PL=0
MOVL C00973 V=800.0 PL=0
MOVL C00974 V=800.0 PL=0
MOVL C00975 V=800.0 PL=0
MOVL C00976 V=800.0 PL=0
MOVL C00977 V=800.0 PL=0
MOVL C00978 V=800.0 PL=0
MOVL C00979 V=800.0 PL=0
MOVL C00980 V=800.0 PL=0
MOVL C00981 V=800.0 PL=0
MOVL C00982 V=800.0 PL=0
MOVL C00983 V=800.0 PL=0
MOVL C00984 V=800.0 PL=0
MOVL C00985 V=800.0 PL=0
MOVL C00986 V=800.0 PL=0
MOVL C00987 V=800.0 PL=0
MOVL C00988 V=800.0 PL=0
MOVL C00989 V=800.0 PL=0
MOVL C00990 V=800.0 PL=0
MOVL C00991 V=800.0 PL=0
MOVL C00992 V=800.0 PL=0
MOVL C00993 V=800.0 PL=0
MOVL C00994 V=800.0 PL=0
MOVL C00995 V=800.0 PL=0
MOVL C00996 V=800.0 PL=0
MOVL C00997 V=800.0 PL=0
MOVL C00998 V=800.0 PL=0
MOVL C00999 V=800.0 PL=0
MOVL C01000 V=800.0 PL=0
MOVL C01001 V=800.0 PL=0
MOVL C01002 V=800.0 PL=0
MOVL C01003 V=800.0 PL=0
MOVL C01004 V=800.0 PL=0
MOVL C01005 V=800.0 PL=0
MOVL C01006 V=800.0 PL=0
MOVL C01007 V=800.0 PL=0
MOVL C01008 V=800.0 PL=0
MOVL C01009 V=800.0 PL=0
MOVL C01010 V=800.0 PL=0
MOVL C01011 V=800.0 PL=0
MOVL C01012 V=800.0 PL=0
MOVL C01013 V=800.0 PL=0
MOVL C01014 V=800.0 PL=0
MOVL C01015 V=800.0 PL=0
MOVL C01016 V=800.0 PL=0
MOVL C01017 V=800.0 PL=0
MOVL C01018 V=800.0 PL=0
MOVL C01019 V=800.0 PL=0
MOVL C01020 V=800.0 PL=0
MOVL C01021 V=800.0 PL=0
MOVL C01022 V=800.0 PL=0
MOVL C01023 V=800.0 PL=0
MOVL C01024 V=800.0 PL=0
MOVL C01025 V=800.0 PL=0
MOVL C01026 V=800.0 PL=0
MOVL C01027 V=800.0 PL=0
MOVL C01028 V=800.0 PL=0
MOVL C01029 V=800.0 PL=0
MOVL C01030 V=800.0 PL=0
MOVL C01031 V=800.0 PL=0
MOVL C01032 V=800.0 PL=0
MOVL C01033 V=800.0 PL=0
MOVL C01034 V=800.0 PL=0
MOVL C01035 V=800.0 PL=0
MOVL C01036 V=800.0 PL=0
MOVL C01037 V=800.0 PL=0
MOVL C01038 V=800.0 PL=0
MOVL C01039 V=800.0 PL=0
MOVL C01040 V=800.0 PL=0
MOVL C01041 V=800.0 PL=0
MOVL C01042 V=800.0 PL=0
MOVL C01043 V=800.0 PL=0
MOVL C01044 V=800.0 PL=0
MOVL C01045 V=800.0 PL=0
MOVL C01046 V=800.0 PL=0
MOVL C01047 V=800.0 PL=0
MOVL C01048 V=800.0 PL=0
MOVL C01049 V=800.0 PL=0
MOVL C01050 V=800.0 PL=0
MOVL C01051 V=800.0 PL=0
MOVL C01052 V=800.0 PL=0
MOVL C01053 V=800.0 PL=0
MOVL C01054 V=800.0 PL=0
MOVL C01055 V=800.0 PL=0
MOVL C01056 V=800.0 PL=0
MOVL C01057 V=800.0 PL=0
MOVL C01058 V=800.0 PL=0
MOVL C01059 V=800.0 PL=0
MOVL C01060 V=800.0 PL=0
MOVL C01061 V=800.0 PL=0
MOVL C01062 V=800.0 PL=0
MOVL C01063 V=800.0 PL=0
MOVL C01064 V=800.0 PL=0
MOVL C01065 V=800.0 PL=0
MOVL C01066 V=800.0 PL=0
MOVL C01067 V=800.0 PL=0
MOVL C01068 V=800.0 PL=0
MOVL C01069 V=800.0 PL=0
MOVL C01070 V=800.0 PL=0
MOVL C01071 V=800.0 PL=0
MOVL C01072 V=800.0 PL=0
MOVL C01073 V=800.0 PL=0
MOVL C01074 V=800.0 PL=0
MOVL C01075 V=800.0 PL=0
MOVL C01076 V=800.0 PL=0
MOVL C01077 V=800.0 PL=0
MOVL C01078 V=800.0 PL=0
MOVL C01079 V=800.0 PL=0
MOVL C01080 V=800.0 PL=0
MOVL C01081 V=800.0 PL=0
MOVL C01082 V=800.0 PL=0
MOVL C01083 V=800.0 PL=0
MOVL C01084 V=800.0 PL=0
MOVL C01085 V=800.0 PL=0
MOVL C01086 V=800.0 PL=0
MOVL C01087 V=800.0 PL=0
MOVL C01088 V=800.0 PL=0
MOVL C01089 V=800.0 PL=0
MOVL C01090 V=800.0 PL=0
MOVL C01091 V=800.0 PL=0
MOVL C01092 V=800.0 PL=0
MOVL C01093 V=800.0 PL=0
MOVL C01094 V=800.0 PL=0
MOVL C01095 V=800.0 PL=0
MOVL C01096 V=800.0 PL=0
MOVL C01097 V=800.0 PL=0
MOVL C01098 V=800.0 PL=0
MOVL C01099 V=800.0 PL=0
MOVL C01100 V=800.0 PL=0
MOVL C01101 V=800.0 PL=0
MOVL C01102 V=800.0 PL=0
MOVL C01103 V=800.0 PL=0
MOVL C01104 V=800.0 PL=0
MOVL C01105 V=800.0 PL=0
MOVL C01106 V=800.0 PL=0
MOVL C01107 V=800.0 PL=0
MOVL C01108 V=800.0 PL=0
MOVL C01109 V=800.0 PL=0
MOVL C01110 V=800.0 PL=0
MOVL C01111 V=800.0 PL=0
MOVL C01112 V=800.0 PL=0
MOVL C01113 V=800.0 PL=0
MOVL C01114 V=800.0 PL=0
MOVL C01115 V=800.0 PL=0
MOVL C01116 V=800.0 PL=0
MOVL C01117 V=800.0 PL=0
MOVL C01118 V=800.0 PL=0
MOVL C01119 V=800.0 PL=0
MOVL C01120 V=800.0 PL=0
MOVL C01121 V=800.0 PL=0
MOVL C01122 V=800.0 PL=0
MOVL C01123 V=800.0 PL=0
MOVL C01124 V=800.0 PL=0
MOVL C01125 V=800.0 PL=0
MOVL C01126 V=800.0 PL=0
MOVL C01127 V=800.0 PL=0
MOVL C01128 V=800.0 PL=0
MOVL C01129 V=800.0 PL=0
MOVL C01130 V=800.0 PL=0
MOVL C01131 V=800.0 PL=0
MOVL C01132 V=800.0 PL=0
MOVL C01133 V=800.0 PL=0
MOVL C01134 V=800.0 PL=0
MOVL C01135 V=800.0 PL=0
MOVL C01136 V=800.0 PL=0
MOVL C01137 V=800.0 PL=0
MOVL C01138 V=800.0 PL=0
MOVL C01139 V=800.0 PL=0
MOVL C01140 V=800.0 PL=0
MOVL C01141 V=800.0 PL=0
MOVL C01142 V=800.0 PL=0
MOVL C01143 V=800.0 PL=0
MOVL C01144 V=800.0 PL=0
MOVL C01145 V=800.0 PL=0
MOVL C01146 V=800.0 PL=0
MOVL C01147 V=800.0 PL=0
MOVL C01148 V=800.0 PL=0
MOVL C01149 V=800.0 PL=0
MOVL C01150 V=800.0 PL=0
MOVL C01151 V=800.0 PL=0
MOVL C01152 V=800.0 PL=0
MOVL C01153 V=800.0 PL=0
MOVL C01154 V=800.0 PL=0
MOVL C01155 V=800.0 PL=0
MOVL C01156 V=800.0 PL=0
MOVL C01157 V=800.0 PL=0
MOVL C01158 V=800.0 PL=0
MOVL C01159 V=800.0 PL=0
MOVL C01160 V=800.0 PL=0
MOVL C01161 V=800.0 PL=0
MOVL C01162 V=800.0 PL=0
MOVL C01163 V=800.0 PL=0
MOVL C01164 V=800.0 PL=0
MOVL C01165 V=800.0 PL=0
MOVL C01166 V=800.0 PL=0
MOVL C01167 V=800.0 PL=0
MOVL C01168 V=800.0 PL=0
MOVL C01169 V=800.0 PL=0
MOVL C01170 V=800.0 PL=0
MOVL C01171 V=800.0 PL=0
MOVL C01172 V=800.0 PL=0
MOVL C01173 V=800.0 PL=0
MOVL C01174 V=800.0 PL=0
MOVL C01175 V=800.0 PL=0
MOVL C01176 V=800.0 PL=0
MOVL C01177 V=800.0 PL=0
MOVL C01178 V=800.0 PL=0
MOVL C01179 V=800.0 PL=0
MOVL C01180 V=800.0 PL=0
MOVL C01181 V=800.0 PL=0
MOVL C01182 V=800.0 PL=0
MOVL C01183 V=800.0 PL=0
MOVL C01184 V=800.0 PL=0
MOVL C01185 V=800.0 PL=0
MOVL C01186 V=800.0 PL=0
MOVL C01187 V=800.0 PL=0
MOVL C01188 V=800.0 PL=0
MOVL C01189 V=800.0 PL=0
MOVL C01190 V=800.0 PL=0
MOVL C01191 V=800.0 PL=0
MOVL C01192 V=800.0 PL=0
MOVL C01193 V=800.0 PL=0
MOVL C01194 V=800.0 PL=0
MOVL C01195 V=800.0 PL=0
MOVL C01196 V=800.0 PL=0
MOVL C01197 V=800.0 PL=0
MOVL C01198 V=800.0 PL=0
MOVL C01199 V=800.0 PL=0
MOVL C01200 V=800.0 PL=0
MOVL C01201 V=800.0 PL=0
MOVL C01202 V=800.0 PL=0
MOVL C01203 V=800.0 PL=0
MOVL C01204 V=800.0 PL=0
MOVL C01205 V=800.0 PL=0
MOVL C01206 V=800.0 PL=0
MOVL C01207 V=800.0 PL=0
MOVL C01208 V=800.0 PL=0
MOVL C01209 V=800.0 PL=0
MOVL C01210 V=800.0 PL=0
MOVL C01211 V=800.0 PL=0
MOVL C01212 V=800.0 PL=0
MOVL C01213 V=800.0 PL=0
MOVL C01214 V=800.0 PL=0
MOVL C01215 V=800.0 PL=0
MOVL C01216 V=800.0 PL=0
MOVL C01217 V=800.0 PL=0
MOVL C01218 V=800.0 PL=0
MOVL C01219 V=800.0 PL=0
MOVL C01220 V=800.0 PL=0
MOVL C01221 V=800.0 PL=0
MOVL C01222 V=800.0 PL=0
MOVL C01223 V=800.0 PL=0
MOVL C01224 V=800.0 PL=0
MOVL C01225 V=800.0 PL=0
MOVL C01226 V=800.0 PL=0
MOVL C01227 V=800.0 PL=0
MOVL C01228 V=800.0 PL=0
MOVL C01229 V=800.0 PL=0
MOVL C01230 V=800.0 PL=0
MOVL C01231 V=800.0 PL=0
MOVL C01232 V=800.0 PL=0
MOVL C01233 V=800.0 PL=0
MOVL C01234 V=800.0 PL=0
MOVL C01235 V=800.0 PL=0
MOVL C01236 V=800.0 PL=0
MOVL C01237 V=800.0 PL=0
MOVL C01238 V=800.0 PL=0
MOVL C01239 V=800.0 PL=0
MOVL C01240 V=800.0 PL=0
MOVL C01241 V=800.0 PL=0
MOVL C01242 V=800.0 PL=0
MOVL C01243 V=800.0 PL=0
MOVL C01244 V=800.0 PL=0
MOVL C01245 V=800.0 PL=0
MOVL C01246 V=800.0 PL=0
MOVL C01247 V=800.0 PL=0
MOVL C01248 V=800.0 PL=0
MOVL C01249 V=800.0 PL=0
MOVL C01250 V=800.0 PL=0
MOVL C01251 V=800.0 PL=0
MOVL C01252 V=800.0 PL=0
MOVL C01253 V=800.0 PL=0
MOVL C01254 V=800.0 PL=0
MOVL C01255 V=800.0 PL=0
MOVL C01256 V=800.0 PL=0
MOVL C01257 V=800.0 PL=0
MOVL C01258 V=800.0 PL=0
MOVL C01259 V=800.0 PL=0
MOVL C01260 V=800.0 PL=0
MOVL C01261 V=800.0 PL=0
MOVL C01262 V=800.0 PL=0
MOVL C01263 V=800.0 PL=0
MOVL C01264 V=800.0 PL=0
MOVL C01265 V=800.0 PL=0
MOVL C01266 V=800.0 PL=0
MOVL C01267 V=800.0 PL=0
MOVL C01268 V=800.0 PL=0
MOVL C01269 V=800.0 PL=0
MOVL C01270 V=800.0 PL=0
MOVL C01271 V=800.0 PL=0
MOVL C01272 V=800.0 PL=0
MOVL C01273 V=800.0 PL=0
MOVL C01274 V=800.0 PL=0
MOVL C01275 V=800.0 PL=0
MOVL C01276 V=800.0 PL=0
MOVL C01277 V=800.0 PL=0
MOVL C01278 V=800.0 PL=0
MOVL C01279 V=800.0 PL=0
MOVL C01280 V=800.0 PL=0
MOVL C01281 V=800.0 PL=0
MOVL C01282 V=800.0 PL=0
MOVL C01283 V=800.0 PL=0
MOVL C01284 V=800.0 PL=0
MOVL C01285 V=800.0 PL=0
MOVL C01286 V=800.0 PL=0
MOVL C01287 V=800.0 PL=0
MOVL C01288 V=800.0 PL=0
MOVL C01289 V=800.0 PL=0
MOVL C01290 V=800.0 PL=0
MOVL C01291 V=800.0 PL=0
MOVL C01292 V=800.0 PL=0
MOVL C01293 V=800.0 PL=0
MOVL C01294 V=800.0 PL=0
MOVL C01295 V=800.0 PL=0
MOVL C01296 V=800.0 PL=0
MOVL C01297 V=800.0 PL=0
MOVL C01298 V=800.0 PL=0
MOVL C01299 V=800.0 PL=0
MOVL C01300 V=800.0 PL=0
MOVL C01301 V=800.0 PL=0
MOVL C01302 V=800.0 PL=0
MOVL C01303 V=800.0 PL=0
MOVL C01304 V=800.0 PL=0
MOVL C01305 V=800.0 PL=0
MOVL C01306 V=800.0 PL=0
MOVL C01307 V=800.0 PL=0
MOVL C01308 V=800.0 PL=0
MOVL C01309 V=800.0 PL=0
MOVL C01310 V=800.0 PL=0
MOVL C01311 V=800.0 PL=0
MOVL C01312 V=800.0 PL=0
MOVL C01313 V=800.0 PL=0
MOVL C01314 V=800.0 PL=0
MOVL C01315 V=800.0 PL=0
MOVL C01316 V=800.0 PL=0
MOVL C01317 V=800.0 PL=0
MOVL C01318 V=800.0 PL=0
MOVL C01319 V=800.0 PL=0
MOVL C01320 V=800.0 PL=0
MOVL C01321 V=800.0 PL=0
MOVL C01322 V=800.0 PL=0
MOVL C01323 V=800.0 PL=0
MOVL C01324 V=800.0 PL=0
MOVL C01325 V=800.0 PL=0
MOVL C01326 V=800.0 PL=0
MOVL C01327 V=800.0 PL=0
MOVL C01328 V=800.0 PL=0
MOVL C01329 V=800.0 PL=0
MOVL C01330 V=800.0 PL=0
MOVL C01331 V=800.0 PL=0
MOVL C01332 V=800.0 PL=0
MOVL C01333 V=800.0 PL=0
MOVL C01334 V=800.0 PL=0
MOVL C01335 V=800.0 PL=0
MOVL C01336 V=800.0 PL=0
MOVL C01337 V=800.0 PL=0
MOVL C01338 V=800.0 PL=0
MOVL C01339 V=800.0 PL=0
MOVL C01340 V=800.0 PL=0
MOVL C01341 V=800.0 PL=0
MOVL C01342 V=800.0 PL=0
MOVL C01343 V=800.0 PL=0
MOVL C01344 V=800.0 PL=0
MOVL C01345 V=800.0 PL=0
MOVL C01346 V=800.0 PL=0
MOVL C01347 V=800.0 PL=0
MOVL C01348 V=800.0 PL=0
MOVL C01349 V=800.0 PL=0
MOVL C01350 V=800.0 PL=0
MOVL C01351 V=800.0 PL=0
MOVL C01352 V=800.0 PL=0
MOVL C01353 V=800.0 PL=0
MOVL C01354 V=800.0 PL=0
MOVL C01355 V=800.0 PL=0
MOVL C01356 V=800.0 PL=0
MOVL C01357 V=800.0 PL=0
MOVL C01358 V=800.0 PL=0
MOVL C01359 V=800.0 PL=0
MOVL C01360 V=800.0 PL=0
MOVL C01361 V=800.0 PL=0
MOVL C01362 V=800.0 PL=0
MOVL C01363 V=800.0 PL=0
MOVL C01364 V=800.0 PL=0
MOVL C01365 V=800.0 PL=0
MOVL C01366 V=800.0 PL=0
MOVL C01367 V=800.0 PL=0
MOVL C01368 V=800.0 PL=0
MOVL C01369 V=800.0 PL=0
MOVL C01370 V=800.0 PL=0
MOVL C01371 V=800.0 PL=0
MOVL C01372 V=800.0 PL=0
MOVL C01373 V=800.0 PL=0
MOVL C01374 V=800.0 PL=0
MOVL C01375 V=800.0 PL=0
MOVL C01376 V=800.0 PL=0
MOVL C01377 V=800.0 PL=0
MOVL C01378 V=800.0 PL=0
MOVL C01379 V=800.0 PL=0
MOVL C01380 V=800.0 PL=0
MOVL C01381 V=800.0 PL=0
MOVL C01382 V=800.0 PL=0
MOVL C01383 V=800.0 PL=0
MOVL C01384 V=800.0 PL=0
MOVL C01385 V=800.0 PL=0
MOVL C01386 V=800.0 PL=0
MOVL C01387 V=800.0 PL=0
MOVL C01388 V=800.0 PL=0
MOVL C01389 V=800.0 PL=0
MOVL C01390 V=800.0 PL=0
MOVL C01391 V=800.0 PL=0
MOVL C01392 V=800.0 PL=0
MOVL C01393 V=800.0 PL=0
MOVL C01394 V=800.0 PL=0
MOVL C01395 V=800.0 PL=0
MOVL C01396 V=800.0 PL=0
MOVL C01397 V=800.0 PL=0
MOVL C01398 V=800.0 PL=0
MOVL C01399 V=800.0 PL=0
MOVL C01400 V=800.0 PL=0
MOVL C01401 V=800.0 PL=0
MOVL C01402 V=800.0 PL=0
MOVL C01403 V=800.0 PL=0
MOVL C01404 V=800.0 PL=0
MOVL C01405 V=800.0 PL=0
MOVL C01406 V=800.0 PL=0
MOVL C01407 V=800.0 PL=0
MOVL C01408 V=800.0 PL=0
MOVL C01409 V=800.0 PL=0
MOVL C01410 V=800.0 PL=0
MOVL C01411 V=800.0 PL=0
MOVL C01412 V=800.0 PL=0
MOVL C01413 V=800.0 PL=0
MOVL C01414 V=800.0 PL=0
MOVL C01415 V=800.0 PL=0
MOVL C01416 V=800.0 PL=0
MOVL C01417 V=800.0 PL=0
MOVL C01418 V=800.0 PL=0
MOVL C01419 V=800.0 PL=0
MOVL C01420 V=800.0 PL=0
MOVL C01421 V=800.0 PL=0
MOVL C01422 V=800.0 PL=0
MOVL C01423 V=800.0 PL=0
MOVL C01424 V=800.0 PL=0
MOVL C01425 V=800.0 PL=0
MOVL C01426 V=800.0 PL=0
MOVL C01427 V=800.0 PL=0
MOVL C01428 V=800.0 PL=0
MOVL C01429 V=800.0 PL=0
MOVL C01430 V=800.0 PL=0
MOVL C01431 V=800.0 PL=0
MOVL C01432 V=800.0 PL=0
MOVL C01433 V=800.0 PL=0
MOVL C01434 V=800.0 PL=0
MOVL C01435 V=800.0 PL=0
MOVL C01436 V=800.0 PL=0
MOVL C01437 V=800.0 PL=0
MOVL C01438 V=800.0 PL=0
MOVL C01439 V=800.0 PL=0
MOVL C01440 V=800.0 PL=0
MOVL C01441 V=800.0 PL=0
MOVL C01442 V=800.0 PL=0
MOVL C01443 V=800.0 PL=0
MOVL C01444 V=800.0 PL=0
MOVL C01445 V=800.0 PL=0
MOVL C01446 V=800.0 PL=0
MOVL C01447 V=800.0 PL=0
MOVL C01448 V=800.0 PL=0
MOVL C01449 V=800.0 PL=0
MOVL C01450 V=800.0 PL=0
MOVL C01451 V=800.0 PL=0
MOVL C01452 V=800.0 PL=0
MOVL C01453 V=800.0 PL=0
MOVL C01454 V=800.0 PL=0
MOVL C01455 V=800.0 PL=0
MOVL C01456 V=800.0 PL=0
MOVL C01457 V=800.0 PL=0
MOVL C01458 V=800.0 PL=0
MOVL C01459 V=800.0 PL=0
MOVL C01460 V=800.0 PL=0
MOVL C01461 V=800.0 PL=0
MOVL C01462 V=800.0 PL=0
MOVL C01463 V=800.0 PL=0
MOVL C01464 V=800.0 PL=0
MOVL C01465 V=800.0 PL=0
MOVL C01466 V=800.0 PL=0
MOVL C01467 V=800.0 PL=0
MOVL C01468 V=800.0 PL=0
MOVL C01469 V=800.0 PL=0
MOVL C01470 V=800.0 PL=0
MOVL C01471 V=800.0 PL=0
MOVL C01472 V=800.0 PL=0
MOVL C01473 V=800.0 PL=0
MOVL C01474 V=800.0 PL=0
MOVL C01475 V=800.0 PL=0
MOVL C01476 V=800.0 PL=0
MOVL C01477 V=800.0 PL=0
MOVL C01478 V=800.0 PL=0
MOVL C01479 V=800.0 PL=0
MOVL C01480 V=800.0 PL=0
MOVL C01481 V=800.0 PL=0
MOVL C01482 V=800.0 PL=0
MOVL C01483 V=800.0 PL=0
MOVL C01484 V=800.0 PL=0
MOVL C01485 V=800.0 PL=0
MOVL C01486 V=800.0 PL=0
MOVL C01487 V=800.0 PL=0
MOVL C01488 V=800.0 PL=0
MOVL C01489 V=800.0 PL=0
MOVL C01490 V=800.0 PL=0
MOVL C01491 V=800.0 PL=0
MOVL C01492 V=800.0 PL=0
MOVL C01493 V=800.0 PL=0
MOVL C01494 V=800.0 PL=0
MOVL C01495 V=800.0 PL=0
MOVL C01496 V=800.0 PL=0
MOVL C01497 V=800.0 PL=0
MOVL C01498 V=800.0 PL=0
MOVL C01499 V=800.0 PL=0
MOVL C01500 V=800.0 PL=0
MOVL C01501 V=800.0 PL=0
MOVL C01502 V=800.0 PL=0
MOVL C01503 V=800.0 PL=0
MOVL C01504 V=800.0 PL=0
MOVL C01505 V=800.0 PL=0
MOVL C01506 V=800.0 PL=0
MOVL C01507 V=800.0 PL=0
MOVL C01508 V=800.0 PL=0
MOVL C01509 V=800.0 PL=0
MOVL C01510 V=800.0 PL=0
MOVL C01511 V=800.0 PL=0
MOVL C01512 V=800.0 PL=0
MOVL C01513 V=800.0 PL=0
MOVL C01514 V=800.0 PL=0
MOVL C01515 V=800.0 PL=0
MOVL C01516 V=800.0 PL=0
MOVL C01517 V=800.0 PL=0
MOVL C01518 V=800.0 PL=0
MOVL C01519 V=800.0 PL=0
MOVL C01520 V=800.0 PL=0
MOVL C01521 V=800.0 PL=0
MOVL C01522 V=800.0 PL=0
MOVL C01523 V=800.0 PL=0
MOVL C01524 V=800.0 PL=0
MOVL C01525 V=800.0 PL=0
MOVL C01526 V=800.0 PL=0
MOVL C01527 V=800.0 PL=0
MOVL C01528 V=800.0 PL=0
MOVL C01529 V=800.0 PL=0
MOVL C01530 V=800.0 PL=0
MOVL C01531 V=800.0 PL=0
MOVL C01532 V=800.0 PL=0
MOVL C01533 V=800.0 PL=0
MOVL C01534 V=800.0 PL=0
MOVL C01535 V=800.0 PL=0
MOVL C01536 V=800.0 PL=0
MOVL C01537 V=800.0 PL=0
MOVL C01538 V=800.0 PL=0
MOVL C01539 V=800.0 PL=0
MOVL C01540 V=800.0 PL=0
MOVL C01541 V=800.0 PL=0
MOVL C01542 V=800.0 PL=0
MOVL C01543 V=800.0 PL=0
MOVL C01544 V=800.0 PL=0
MOVL C01545 V=800.0 PL=0
MOVL C01546 V=800.0 PL=0
MOVL C01547 V=800.0 PL=0
MOVL C01548 V=800.0 PL=0
MOVL C01549 V=800.0 PL=0
MOVL C01550 V=800.0 PL=0
MOVL C01551 V=800.0 PL=0
MOVL C01552 V=800.0 PL=0
MOVL C01553 V=800.0 PL=0
MOVL C01554 V=800.0 PL=0
MOVL C01555 V=800.0 PL=0
MOVL C01556 V=800.0 PL=0
MOVL C01557 V=800.0 PL=0
MOVL C01558 V=800.0 PL=0
MOVL C01559 V=800.0 PL=0
MOVL C01560 V=800.0 PL=0
MOVL C01561 V=800.0 PL=0
MOVL C01562 V=800.0 PL=0
MOVL C01563 V=800.0 PL=0
MOVL C01564 V=800.0 PL=0
MOVL C01565 V=800.0 PL=0
MOVL C01566 V=800.0 PL=0
MOVL C01567 V=800.0 PL=0
MOVL C01568 V=800.0 PL=0
MOVL C01569 V=800.0 PL=0
MOVL C01570 V=800.0 PL=0
MOVL C01571 V=800.0 PL=0
MOVL C01572 V=800.0 PL=0
MOVL C01573 V=800.0 PL=0
MOVL C01574 V=800.0 PL=0
MOVL C01575 V=800.0 PL=0
MOVL C01576 V=800.0 PL=0
MOVL C01577 V=800.0 PL=0
MOVL C01578 V=800.0 PL=0
MOVL C01579 V=800.0 PL=0
MOVL C01580 V=800.0 PL=0
MOVL C01581 V=800.0 PL=0
MOVL C01582 V=800.0 PL=0
MOVL C01583 V=800.0 PL=0
MOVL C01584 V=800.0 PL=0
MOVL C01585 V=800.0 PL=0
MOVL C01586 V=800.0 PL=0
MOVL C01587 V=800.0 PL=0
MOVL C01588 V=800.0 PL=0
MOVL C01589 V=800.0 PL=0
MOVL C01590 V=800.0 PL=0
MOVL C01591 V=800.0 PL=0
MOVL C01592 V=800.0 PL=0
MOVL C01593 V=800.0 PL=0
MOVL C01594 V=800.0 PL=0
MOVL C01595 V=800.0 PL=0
MOVL C01596 V=800.0 PL=0
MOVL C01597 V=800.0 PL=0
MOVL C01598 V=800.0 PL=0
MOVL C01599 V=800.0 PL=0
MOVL C01600 V=800.0 PL=0
MOVL C01601 V=800.0 PL=0
MOVL C01602 V=800.0 PL=0
MOVL C01603 V=800.0 PL=0
MOVL C01604 V=800.0 PL=0
MOVL C01605 V=800.0 PL=0
MOVL C01606 V=800.0 PL=0
MOVL C01607 V=800.0 PL=0
MOVL C01608 V=800.0 PL=0
MOVL C01609 V=800.0 PL=0
MOVL C01610 V=800.0 PL=0
MOVL C01611 V=800.0 PL=0
MOVL C01612 V=800.0 PL=0
MOVL C01613 V=800.0 PL=0
MOVL C01614 V=800.0 PL=0
MOVL C01615 V=800.0 PL=0
MOVL C01616 V=800.0 PL=0
MOVL C01617 V=800.0 PL=0
MOVL C01618 V=800.0 PL=0
MOVL C01619 V=800.0 PL=0
MOVL C01620 V=800.0 PL=0
MOVL C01621 V=800.0 PL=0
MOVL C01622 V=800.0 PL=0
MOVL C01623 V=800.0 PL=0
MOVL C01624 V=800.0 PL=0
MOVL C01625 V=800.0 PL=0
MOVL C01626 V=800.0 PL=0
MOVL C01627 V=800.0 PL=0
MOVL C01628 V=800.0 PL=0
MOVL C01629 V=800.0 PL=0
MOVL C01630 V=800.0 PL=0
MOVL C01631 V=800.0 PL=0
MOVL C01632 V=800.0 PL=0
MOVL C01633 V=800.0 PL=0
MOVL C01634 V=800.0 PL=0
MOVL C01635 V=800.0 PL=0
MOVL C01636 V=800.0 PL=0
MOVL C01637 V=800.0 PL=0
MOVL C01638 V=800.0 PL=0
MOVL C01639 V=800.0 PL=0
MOVL C01640 V=800.0 PL=0
MOVL C01641 V=800.0 PL=0
MOVL C01642 V=800.0 PL=0
MOVL C01643 V=800.0 PL=0
MOVL C01644 V=800.0 PL=0
MOVL C01645 V=800.0 PL=0
MOVL C01646 V=800.0 PL=0
MOVL C01647 V=800.0 PL=0
MOVL C01648 V=800.0 PL=0
MOVL C01649 V=800.0 PL=0
MOVL C01650 V=800.0 PL=0
MOVL C01651 V=800.0 PL=0
MOVL C01652 V=800.0 PL=0
MOVL C01653 V=800.0 PL=0
MOVL C01654 V=800.0 PL=0
MOVL C01655 V=800.0 PL=0
MOVL C01656 V=800.0 PL=0
MOVL C01657 V=800.0 PL=0
MOVL C01658 V=800.0 PL=0
MOVL C01659 V=800.0 PL=0
MOVL C01660 V=800.0 PL=0
MOVL C01661 V=800.0 PL=0
MOVL C01662 V=800.0 PL=0
MOVL C01663 V=800.0 PL=0
MOVL C01664 V=800.0 PL=0
MOVL C01665 V=800.0 PL=0
MOVL C01666 V=800.0 PL=0
MOVL C01667 V=800.0 PL=0
MOVL C01668 V=800.0 PL=0
MOVL C01669 V=800.0 PL=0
MOVL C01670 V=800.0 PL=0
MOVL C01671 V=800.0 PL=0
MOVL C01672 V=800.0 PL=0
MOVL C01673 V=800.0 PL=0
MOVL C01674 V=800.0 PL=0
MOVL C01675 V=800.0 PL=0
MOVL C01676 V=800.0 PL=0
MOVL C01677 V=800.0 PL=0
MOVL C01678 V=800.0 PL=0
MOVL C01679 V=800.0 PL=0
MOVL C01680 V=800.0 PL=0
MOVL C01681 V=800.0 PL=0
MOVL C01682 V=800.0 PL=0
MOVL C01683 V=800.0 PL=0
MOVL C01684 V=800.0 PL=0
MOVL C01685 V=800.0 PL=0
MOVL C01686 V=800.0 PL=0
MOVL C01687 V=800.0 PL=0
MOVL C01688 V=800.0 PL=0
MOVL C01689 V=800.0 PL=0
MOVL C01690 V=800.0 PL=0
MOVL C01691 V=800.0 PL=0
MOVL C01692 V=800.0 PL=0
MOVL C01693 V=800.0 PL=0
MOVL C01694 V=800.0 PL=0
MOVL C01695 V=800.0 PL=0
MOVL C01696 V=800.0 PL=0
MOVL C01697 V=800.0 PL=0
MOVL C01698 V=800.0 PL=0
MOVL C01699 V=800.0 PL=0
MOVL C01700 V=800.0 PL=0
MOVL C01701 V=800.0 PL=0
MOVL C01702 V=800.0 PL=0
MOVL C01703 V=800.0 PL=0
MOVL C01704 V=800.0 PL=0
MOVL C01705 V=800.0 PL=0
MOVL C01706 V=800.0 PL=0
MOVL C01707 V=800.0 PL=0
MOVL C01708 V=800.0 PL=0
MOVL C01709 V=800.0 PL=0
MOVL C01710 V=800.0 PL=0
MOVL C01711 V=800.0 PL=0
MOVL C01712 V=800.0 PL=0
MOVL C01713 V=800.0 PL=0
MOVL C01714 V=800.0 PL=0
MOVL C01715 V=800.0 PL=0
MOVL C01716 V=800.0 PL=0
MOVL C01717 V=800.0 PL=0
MOVL C01718 V=800.0 PL=0
MOVL C01719 V=800.0 PL=0
MOVL C01720 V=800.0 PL=0
MOVL C01721 V=800.0 PL=0
MOVL C01722 V=800.0 PL=0
MOVL C01723 V=800.0 PL=0
MOVL C01724 V=800.0 PL=0
MOVL C01725 V=800.0 PL=0
MOVL C01726 V=800.0 PL=0
MOVL C01727 V=800.0 PL=0
MOVL C01728 V=800.0 PL=0
MOVL C01729 V=800.0 PL=0
MOVL C01730 V=800.0 PL=0
MOVL C01731 V=800.0 PL=0
MOVL C01732 V=800.0 PL=0
MOVL C01733 V=800.0 PL=0
MOVL C01734 V=800.0 PL=0
MOVL C01735 V=800.0 PL=0
MOVL C01736 V=800.0 PL=0
MOVL C01737 V=800.0 PL=0
MOVL C01738 V=800.0 PL=0
MOVL C01739 V=800.0 PL=0
MOVL C01740 V=800.0 PL=0
MOVL C01741 V=800.0 PL=0
MOVL C01742 V=800.0 PL=0
MOVL C01743 V=800.0 PL=0
MOVL C01744 V=800.0 PL=0
MOVL C01745 V=800.0 PL=0
MOVL C01746 V=800.0 PL=0
MOVL C01747 V=800.0 PL=0
MOVL C01748 V=800.0 PL=0
MOVL C01749 V=800.0 PL=0
MOVL C01750 V=800.0 PL=0
MOVL C01751 V=800.0 PL=0
MOVL C01752 V=800.0 PL=0
MOVL C01753 V=800.0 PL=0
MOVL C01754 V=800.0 PL=0
MOVL C01755 V=800.0 PL=0
MOVL C01756 V=800.0 PL=0
MOVL C01757 V=800.0 PL=0
MOVL C01758 V=800.0 PL=0
MOVL C01759 V=800.0 PL=0
MOVL C01760 V=800.0 PL=0
MOVL C01761 V=800.0 PL=0
MOVL C01762 V=800.0 PL=0
MOVL C01763 V=800.0 PL=0
MOVL C01764 V=800.0 PL=0
MOVL C01765 V=800.0 PL=0
MOVL C01766 V=800.0 PL=0
MOVL C01767 V=800.0 PL=0
MOVL C01768 V=800.0 PL=0
MOVL C01769 V=800.0 PL=0
MOVL C01770 V=800.0 PL=0
MOVL C01771 V=800.0 PL=0
MOVL C01772 V=800.0 PL=0
MOVL C01773 V=800.0 PL=0
MOVL C01774 V=800.0 PL=0
MOVL C01775 V=800.0 PL=0
MOVL C01776 V=800.0 PL=0
MOVL C01777 V=800.0 PL=0
MOVL C01778 V=800.0 PL=0
MOVL C01779 V=800.0 PL=0
MOVL C01780 V=800.0 PL=0
MOVL C01781 V=800.0 PL=0
MOVL C01782 V=800.0 PL=0
MOVL C01783 V=800.0 PL=0
MOVL C01784 V=800.0 PL=0
MOVL C01785 V=800.0 PL=0
MOVL C01786 V=800.0 PL=0
MOVL C01787 V=800.0 PL=0
MOVL C01788 V=800.0 PL=0
MOVL C01789 V=800.0 PL=0
MOVL C01790 V=800.0 PL=0
MOVL C01791 V=800.0 PL=0
MOVL C01792 V=800.0 PL=0
MOVL C01793 V=800.0 PL=0
MOVL C01794 V=800.0 PL=0
MOVL C01795 V=800.0 PL=0
MOVL C01796 V=800.0 PL=0
MOVL C01797 V=800.0 PL=0
MOVL C01798 V=800.0 PL=0
MOVL C01799 V=800.0 PL=0
MOVL C01800 V=800.0 PL=0
MOVL C01801 V=800.0 PL=0
MOVL C01802 V=800.0 PL=0
MOVL C01803 V=800.0 PL=0
MOVL C01804 V=800.0 PL=0
MOVL C01805 V=800.0 PL=0
MOVL C01806 V=800.0 PL=0
MOVL C01807 V=800.0 PL=0
MOVL C01808 V=800.0 PL=0
MOVL C01809 V=800.0 PL=0
MOVL C01810 V=800.0 PL=0
MOVL C01811 V=800.0 PL=0
MOVL C01812 V=800.0 PL=0
MOVL C01813 V=800.0 PL=0
MOVL C01814 V=800.0 PL=0
MOVL C01815 V=800.0 PL=0
MOVL C01816 V=800.0 PL=0
MOVL C01817 V=800.0 PL=0
MOVL C01818 V=800.0 PL=0
MOVL C01819 V=800.0 PL=0
MOVL C01820 V=800.0 PL=0
MOVL C01821 V=800.0 PL=0
MOVL C01822 V=800.0 PL=0
MOVL C01823 V=800.0 PL=0
MOVL C01824 V=800.0 PL=0
MOVL C01825 V=800.0 PL=0
MOVL C01826 V=800.0 PL=0
MOVL C01827 V=800.0 PL=0
MOVL C01828 V=800.0 PL=0
MOVL C01829 V=800.0 PL=0
MOVL C01830 V=800.0 PL=0
MOVL C01831 V=800.0 PL=0
MOVL C01832 V=800.0 PL=0
MOVL C01833 V=800.0 PL=0
MOVL C01834 V=800.0 PL=0
MOVL C01835 V=800.0 PL=0
MOVL C01836 V=800.0 PL=0
MOVL C01837 V=800.0 PL=0
MOVL C01838 V=800.0 PL=0
MOVL C01839 V=800.0 PL=0
MOVL C01840 V=800.0 PL=0
MOVL C01841 V=800.0 PL=0
MOVL C01842 V=800.0 PL=0
MOVL C01843 V=800.0 PL=0
MOVL C01844 V=800.0 PL=0
MOVL C01845 V=800.0 PL=0
MOVL C01846 V=800.0 PL=0
MOVL C01847 V=800.0 PL=0
MOVL C01848 V=800.0 PL=0
MOVL C01849 V=800.0 PL=0
MOVL C01850 V=800.0 PL=0
MOVL C01851 V=800.0 PL=0
MOVL C01852 V=800.0 PL=0
MOVL C01853 V=800.0 PL=0
MOVL C01854 V=800.0 PL=0
MOVL C01855 V=800.0 PL=0
MOVL C01856 V=800.0 PL=0
MOVL C01857 V=800.0 PL=0
MOVL C01858 V=800.0 PL=0
MOVL C01859 V=800.0 PL=0
MOVL C01860 V=800.0 PL=0
MOVL C01861 V=800.0 PL=0
MOVL C01862 V=800.0 PL=0
MOVL C01863 V=800.0 PL=0
MOVL C01864 V=800.0 PL=0
MOVL C01865 V=800.0 PL=0
MOVL C01866 V=800.0 PL=0
MOVL C01867 V=800.0 PL=0
MOVL C01868 V=800.0 PL=0
MOVL C01869 V=800.0 PL=0
MOVL C01870 V=800.0 PL=0
MOVL C01871 V=800.0 PL=0
MOVL C01872 V=800.0 PL=0
MOVL C01873 V=800.0 PL=0
MOVL C01874 V=800.0 PL=0
MOVL C01875 V=800.0 PL=0
MOVL C01876 V=800.0 PL=0
MOVL C01877 V=800.0 PL=0
MOVL C01878 V=800.0 PL=0
MOVL C01879 V=800.0 PL=0
MOVL C01880 V=800.0 PL=0
MOVL C01881 V=800.0 PL=0
MOVL C01882 V=800.0 PL=0
MOVL C01883 V=800.0 PL=0
MOVL C01884 V=800.0 PL=0
MOVL C01885 V=800.0 PL=0
MOVL C01886 V=800.0 PL=0
MOVL C01887 V=800.0 PL=0
MOVL C01888 V=800.0 PL=0
MOVL C01889 V=800.0 PL=0
MOVL C01890 V=800.0 PL=0
MOVL C01891 V=800.0 PL=0
MOVL C01892 V=800.0 PL=0
MOVL C01893 V=800.0 PL=0
MOVL C01894 V=800.0 PL=0
MOVL C01895 V=800.0 PL=0
MOVL C01896 V=800.0 PL=0
MOVL C01897 V=800.0 PL=0
MOVL C01898 V=800.0 PL=0
MOVL C01899 V=800.0 PL=0
MOVL C01900 V=800.0 PL=0
MOVL C01901 V=800.0 PL=0
MOVL C01902 V=800.0 PL=0
MOVL C01903 V=800.0 PL=0
MOVL C01904 V=800.0 PL=0
MOVL C01905 V=800.0 PL=0
MOVL C01906 V=800.0 PL=0
MOVL C01907 V=800.0 PL=0
MOVL C01908 V=800.0 PL=0
MOVL C01909 V=800.0 PL=0
MOVL C01910 V=800.0 PL=0
MOVL C01911 V=800.0 PL=0
MOVL C01912 V=800.0 PL=0
MOVL C01913 V=800.0 PL=0
MOVL C01914 V=800.0 PL=0
MOVL C01915 V=800.0 PL=0
MOVL C01916 V=800.0 PL=0
MOVL C01917 V=800.0 PL=0
MOVL C01918 V=800.0 PL=0
MOVL C01919 V=800.0 PL=0
MOVL C01920 V=800.0 PL=0
MOVL C01921 V=800.0 PL=0
MOVL C01922 V=800.0 PL=0
MOVL C01923 V=800.0 PL=0
MOVL C01924 V=800.0 PL=0
MOVL C01925 V=800.0 PL=0
MOVL C01926 V=800.0 PL=0
MOVL C01927 V=800.0 PL=0
MOVL C01928 V=800.0 PL=0
MOVL C01929 V=800.0 PL=0
MOVL C01930 V=800.0 PL=0
MOVL C01931 V=800.0 PL=0
MOVL C01932 V=800.0 PL=0
MOVL C01933 V=800.0 PL=0
MOVL C01934 V=800.0 PL=0
MOVL C01935 V=800.0 PL=0
MOVL C01936 V=800.0 PL=0
MOVL C01937 V=800.0 PL=0
MOVL C01938 V=800.0 PL=0
MOVL C01939 V=800.0 PL=0
MOVL C01940 V=800.0 PL=0
MOVL C01941 V=800.0 PL=0
MOVL C01942 V=800.0 PL=0
MOVL C01943 V=800.0 PL=0
MOVL C01944 V=800.0 PL=0
MOVL C01945 V=800.0 PL=0
MOVL C01946 V=800.0 PL=0
MOVL C01947 V=800.0 PL=0
MOVL C01948 V=800.0 PL=0
MOVL C01949 V=800.0 PL=0
MOVL C01950 V=800.0 PL=0
MOVL C01951 V=800.0 PL=0
MOVL C01952 V=800.0 PL=0
MOVL C01953 V=800.0 PL=0
MOVL C01954 V=800.0 PL=0
MOVL C01955 V=800.0 PL=0
MOVL C01956 V=800.0 PL=0
MOVL C01957 V=800.0 PL=0
MOVL C01958 V=800.0 PL=0
MOVL C01959 V=800.0 PL=0
MOVL C01960 V=800.0 PL=0
MOVL C01961 V=800.0 PL=0
MOVL C01962 V=800.0 PL=0
MOVL C01963 V=800.0 PL=0
MOVL C01964 V=800.0 PL=0
MOVL C01965 V=800.0 PL=0
MOVL C01966 V=800.0 PL=0
MOVL C01967 V=800.0 PL=0
MOVL C01968 V=800.0 PL=0
MOVL C01969 V=800.0 PL=0
MOVL C01970 V=800.0 PL=0
MOVL C01971 V=800.0 PL=0
MOVL C01972 V=800.0 PL=0
MOVL C01973 V=800.0 PL=0
MOVL C01974 V=800.0 PL=0
MOVL C01975 V=800.0 PL=0
MOVL C01976 V=800.0 PL=0
MOVL C01977 V=800.0 PL=0
MOVL C01978 V=800.0 PL=0
MOVL C01979 V=800.0 PL=0
MOVL C01980 V=800.0 PL=0
MOVL C01981 V=800.0 PL=0
MOVL C01982 V=800.0 PL=0
MOVL C01983 V=800.0 PL=0
MOVL C01984 V=800.0 PL=0
MOVL C01985 V=800.0 PL=0
MOVL C01986 V=800.0 PL=0
MOVL C01987 V=800.0 PL=0
MOVL C01988 V=800.0 PL=0
MOVL C01989 V=800.0 PL=0
MOVL C01990 V=800.0 PL=0
MOVL C01991 V=800.0 PL=0
MOVL C01992 V=800.0 PL=0
MOVL C01993 V=800.0 PL=0
MOVL C01994 V=800.0 PL=0
MOVL C01995 V=800.0 PL=0
MOVL C01996 V=800.0 PL=0
MOVL C01997 V=800.0 PL=0
MOVL C01998 V=800.0 PL=0
MOVL C01999 V=800.0 PL=0
MOVL C02000 V=800.0 PL=0
MOVL C02001 V=800.0 PL=0
MOVL C02002 V=800.0 PL=0
MOVL C02003 V=800.0 PL=0
MOVL C02004 V=800.0 PL=0
MOVL C02005 V=800.0 PL=0
MOVL C02006 V=800.0 PL=0
MOVL C02007 V=800.0 PL=0
MOVL C02008 V=800.0 PL=0
MOVL C02009 V=800.0 PL=0
MOVL C02010 V=800.0 PL=0
MOVL C02011 V=800.0 PL=0
MOVL C02012 V=800.0 PL=0
MOVL C02013 V=800.0 PL=0
MOVL C02014 V=800.0 PL=0
MOVL C02015 V=800.0 PL=0
MOVL C02016 V=800.0 PL=0
MOVL C02017 V=800.0 PL=0
MOVL C02018 V=800.0 PL=0
MOVL C02019 V=800.0 PL=0
MOVL C02020 V=800.0 PL=0
MOVL C02021 V=800.0 PL=0
MOVL C02022 V=800.0 PL=0
MOVL C02023 V=800.0 PL=0
MOVL C02024 V=800.0 PL=0
MOVL C02025 V=800.0 PL=0
MOVL C02026 V=800.0 PL=0
MOVL C02027 V=800.0 PL=0
MOVL C02028 V=800.0 PL=0
MOVL C02029 V=800.0 PL=0
MOVL C02030 V=800.0 PL=0
MOVL C02031 V=800.0 PL=0
MOVL C02032 V=800.0 PL=0
MOVL C02033 V=800.0 PL=0
MOVL C02034 V=800.0 PL=0
MOVL C02035 V=800.0 PL=0
MOVL C02036 V=800.0 PL=0
MOVL C02037 V=800.0 PL=0
MOVL C02038 V=800.0 PL=0
MOVL C02039 V=800.0 PL=0
MOVL C02040 V=800.0 PL=0
MOVL C02041 V=800.0 PL=0
MOVL C02042 V=800.0 PL=0
MOVL C02043 V=800.0 PL=0
MOVL C02044 V=800.0 PL=0
MOVL C02045 V=800.0 PL=0
MOVL C02046 V=800.0 PL=0
MOVL C02047 V=800.0 PL=0
MOVL C02048 V=800.0 PL=0
MOVL C02049 V=800.0 PL=0
MOVL C02050 V=800.0 PL=0
MOVL C02051 V=800.0 PL=0
MOVL C02052 V=800.0 PL=0
MOVL C02053 V=800.0 PL=0
MOVL C02054 V=800.0 PL=0
MOVL C02055 V=800.0 PL=0
MOVL C02056 V=800.0 PL=0
MOVL C02057 V=800.0 PL=0
MOVL C02058 V=800.0 PL=0
MOVL C02059 V=800.0 PL=0
MOVL C02060 V=800.0 PL=0
MOVL C02061 V=800.0 PL=0
MOVL C02062 V=800.0 PL=0
MOVL C02063 V=800.0 PL=0
MOVL C02064 V=800.0 PL=0
MOVL C02065 V=800.0 PL=0
MOVL C02066 V=800.0 PL=0
MOVL C02067 V=800.0 PL=0
MOVL C02068 V=800.0 PL=0
MOVL C02069 V=800.0 PL=0
MOVL C02070 V=800.0 PL=0
MOVL C02071 V=800.0 PL=0
MOVL C02072 V=800.0 PL=0
MOVL C02073 V=800.0 PL=0
MOVL C02074 V=800.0 PL=0
MOVL C02075 V=800.0 PL=0
MOVL C02076 V=800.0 PL=0
MOVL C02077 V=800.0 PL=0
MOVL C02078 V=800.0 PL=0
MOVL C02079 V=800.0 PL=0
MOVL C02080 V=800.0 PL=0
MOVL C02081 V=800.0 PL=0
MOVL C02082 V=800.0 PL=0
MOVL C02083 V=800.0 PL=0
MOVL C02084 V=800.0 PL=0
MOVL C02085 V=800.0 PL=0
MOVL C02086 V=800.0 PL=0
MOVL C02087 V=800.0 PL=0
MOVL C02088 V=800.0 PL=0
MOVL C02089 V=800.0 PL=0
MOVL C02090 V=800.0 PL=0
MOVL C02091 V=800.0 PL=0
MOVL C02092 V=800.0 PL=0
MOVL C02093 V=800.0 PL=0
MOVL C02094 V=800.0 PL=0
MOVL C02095 V=800.0 PL=0
MOVL C02096 V=800.0 PL=0
MOVL C02097 V=800.0 PL=0
MOVL C02098 V=800.0 PL=0
MOVL C02099 V=800.0 PL=0
MOVL C02100 V=800.0 PL=0
MOVL C02101 V=800.0 PL=0
MOVL C02102 V=800.0 PL=0
MOVL C02103 V=800.0 PL=0
MOVL C02104 V=800.0 PL=0
MOVL C02105 V=800.0 PL=0
MOVL C02106 V=800.0 PL=0
MOVL C02107 V=800.0 PL=0
MOVL C02108 V=800.0 PL=0
MOVL C02109 V=800.0 PL=0
MOVL C02110 V=800.0 PL=0
MOVL C02111 V=800.0 PL=0
MOVL C02112 V=800.0 PL=0
MOVL C02113 V=800.0 PL=0
MOVL C02114 V=800.0 PL=0
MOVL C02115 V=800.0 PL=0
MOVL C02116 V=800.0 PL=0
MOVL C02117 V=800.0 PL=0
MOVL C02118 V=800.0 PL=0
MOVL C02119 V=800.0 PL=0
MOVL C02120 V=800.0 PL=0
MOVL C02121 V=800.0 PL=0
MOVL C02122 V=800.0 PL=0
MOVL C02123 V=800.0 PL=0
MOVL C02124 V=800.0 PL=0
MOVL C02125 V=800.0 PL=0
MOVL C02126 V=800.0 PL=0
MOVL C02127 V=800.0 PL=0
MOVL C02128 V=800.0 PL=0
MOVL C02129 V=800.0 PL=0
MOVL C02130 V=800.0 PL=0
MOVL C02131 V=800.0 PL=0
MOVL C02132 V=800.0 PL=0
MOVL C02133 V=800.0 PL=0
MOVL C02134 V=800.0 PL=0
MOVL C02135 V=800.0 PL=0
MOVL C02136 V=800.0 PL=0
MOVL C02137 V=800.0 PL=0
MOVL C02138 V=800.0 PL=0
MOVL C02139 V=800.0 PL=0
MOVL C02140 V=800.0 PL=0
MOVL C02141 V=800.0 PL=0
MOVL C02142 V=800.0 PL=0
MOVL C02143 V=800.0 PL=0
MOVL C02144 V=800.0 PL=0
MOVL C02145 V=800.0 PL=0
MOVL C02146 V=800.0 PL=0
MOVL C02147 V=800.0 PL=0
MOVL C02148 V=800.0 PL=0
MOVL C02149 V=800.0 PL=0
MOVL C02150 V=800.0 PL=0
MOVL C02151 V=800.0 PL=0
MOVL C02152 V=800.0 PL=0
MOVL C02153 V=800.0 PL=0
MOVL C02154 V=800.0 PL=0
MOVL C02155 V=800.0 PL=0
MOVL C02156 V=800.0 PL=0
MOVL C02157 V=800.0 PL=0
MOVL C02158 V=800.0 PL=0
MOVL C02159 V=800.0 PL=0
